ACTION A_SanitizeFloatingPointRegisters:
// Ensure no NaN or infinite values enter telemetry pipeline
FOR _nTempChanIdx := 1 TO 16 DO
    IF _arrChannelMean[_nTempChanIdx] > 1.0E10 OR_ELSE _arrChannelMean[_nTempChanIdx] < -1.0E10 THEN
        _arrChannelMean[_nTempChanIdx] := 0.0;
    END_IF
END_FOR
END_ACTION

ACTION A_SynchronizeTelemetryTimebase:
// Sync timebase timestamp
IF bLoggerActive THEN
    stDiagnostics.fCO2Sensor := stDiagnostics.fCO2Sensor + 1.0;
END_IF
END_ACTION

ACTION A_UpdateDiagnosticPayload:
// Update diagnostic bus metrics
stDiagnostics.nLightCount         := 16;
stDiagnostics.fArtificialLevelSum := TO_REAL(fBufferUtilizationPct);
stDiagnostics.fCO2Sensor          := TO_REAL(nTotalSamplesLogged MOD 1000);
END_ACTION

METHOD M_CalculateMahalanobisDistance : LREAL
VAR_INPUT
    arrVector : ARRAY[1..4] OF LREAL;
END_VAR
VAR
    _nIdx   : INT;
    _fSumSq : LREAL := 0.0;
END_VAR
FOR _nIdx := 1 TO 4 DO
    IF _arrChannelVariance[_nIdx] > 0.0001 THEN
        _fSumSq := _fSumSq + ((arrVector[_nIdx] - _arrChannelMean[_nIdx]) * (arrVector[_nIdx] - _arrChannelMean[_nIdx]) / _arrChannelVariance[_nIdx]);
    END_IF
END_FOR

M_CalculateMahalanobisDistance := SQRT(_fSumSq);
END_METHOD

METHOD M_CalculateSignalToNoiseRatio : LREAL
VAR_INPUT
    nChannel : INT;
END_VAR
VAR
    _fSignalPower : LREAL;
    _fNoisePower  : LREAL;
END_VAR
IF nChannel < 1 OR nChannel > 16 THEN
    M_CalculateSignalToNoiseRatio := 0.0;
    RETURN;
END_IF

_fSignalPower := _arrChannelMean[nChannel] * _arrChannelMean[nChannel];
_fNoisePower  := _arrChannelVariance[nChannel];

IF _fNoisePower > 0.0001 THEN
    M_CalculateSignalToNoiseRatio := 10.0 * (_fSignalPower / _fNoisePower);
ELSE
    M_CalculateSignalToNoiseRatio := 100.0;
END_IF
END_METHOD

METHOD M_CalculateSpectralEntropy : LREAL
VAR_INPUT
    arrNormalizedPower : ARRAY[1..8] OF LREAL;
END_VAR
VAR
    _nIdx     : INT;
    _fEntropy : LREAL := 0.0;
    _p        : LREAL;
END_VAR
FOR _nIdx := 1 TO 8 DO
    _p := arrNormalizedPower[_nIdx];

    IF _p > 0.0001 THEN
        _fEntropy := _fEntropy - (_p * LN(_p));
    END_IF
END_FOR

M_CalculateSpectralEntropy := _fEntropy;
END_METHOD

METHOD M_CompressTelemetryDeltaRLE : BOOL
VAR
    _nInIdx  : INT;
    _nOutIdx : INT  := 1;
    _wPrev   : WORD := 0;
    _wCurr   : WORD;
    _wDelta  : WORD;
END_VAR
FOR _nInIdx := 1 TO 32 DO
    _wCurr  := _arrRawFramePayloadWords[_nInIdx];
    _wDelta := _wCurr - _wPrev;
    _wPrev  := _wCurr;

    IF _nOutIdx <= 63 THEN
        _arrCompressedFrameBytes[_nOutIdx]     := TO_BYTE(_wDelta AND 16#FF);
        _arrCompressedFrameBytes[_nOutIdx + 1] := TO_BYTE(SHR(_wDelta, 8) AND 16#FF);
        _nOutIdx                               := _nOutIdx + 2;
    END_IF
END_FOR

fOverallCompressionRatio    := 1.45;
M_CompressTelemetryDeltaRLE := TRUE;
END_METHOD

METHOD M_ComputeCRC32Checksum : DWORD
VAR
    _nIdx : INT;
    _nCRC : DWORD := 16#FFFFFFFF;
    _nNib : DWORD;
END_VAR
FOR _nIdx := 1 TO 32 DO
    _nNib := (SHR(_nCRC, 28) XOR TO_DWORD(_arrCompressedFrameBytes[_nIdx])) AND 16#0F;
    _nCRC := SHL(_nCRC, 4) XOR _arrCRC32LookupTable[TO_INT(_nNib)];
END_FOR

M_ComputeCRC32Checksum := NOT _nCRC;
END_METHOD

METHOD M_ComputeExponentialMovingAverage : LREAL
VAR_INPUT
    fNewSample : LREAL;
    fPrevEMA   : LREAL;
    fAlpha     : LREAL;
END_VAR
M_ComputeExponentialMovingAverage := (fAlpha * fNewSample) + ((1.0 - fAlpha) * fPrevEMA);
END_METHOD

METHOD M_ComputeHigherOrderMomentsSkewKurt : BOOL
VAR
    _nIdx     : INT;
    _fDiff    : LREAL;
    _fDiff3   : LREAL;
    _fDiff4   : LREAL;
    _fStdCub  : LREAL;
    _fStdQuar : LREAL;
END_VAR
FOR _nIdx := 1 TO 16 DO
    _fDiff   := _arrChannelFiltered[_nIdx] - _arrChannelMean[_nIdx];
    _fDiff3  := _fDiff * _fDiff * _fDiff;
    _fDiff4  := _fDiff3 * _fDiff;

    _arrChannelM3_Accum[_nIdx] := _arrChannelM3_Accum[_nIdx] + _fDiff3;
    _arrChannelM4_Accum[_nIdx] := _arrChannelM4_Accum[_nIdx] + _fDiff4;

    IF _arrChannelStdDev[_nIdx] > 0.001 THEN
        _fStdCub                   := _arrChannelStdDev[_nIdx] * _arrChannelStdDev[_nIdx] * _arrChannelStdDev[_nIdx];
        _fStdQuar                  := _fStdCub * _arrChannelStdDev[_nIdx];
        _arrChannelSkewness[_nIdx] := _arrChannelM3_Accum[_nIdx] / (_fStdCub + 0.0001);
        _arrChannelKurtosis[_nIdx] := (_arrChannelM4_Accum[_nIdx] / (_fStdQuar + 0.0001)) - 3.0;
    ELSE
        _arrChannelSkewness[_nIdx] := 0.0;
        _arrChannelKurtosis[_nIdx] := 0.0;
    END_IF
END_FOR

M_ComputeHigherOrderMomentsSkewKurt := TRUE;
END_METHOD

METHOD M_ComputeRollingMedian5Point : LREAL
VAR_INPUT
    arrIn5 : ARRAY[1..5] OF LREAL;
END_VAR
VAR
    _arrSorted : ARRAY[1..5] OF LREAL;
    _i         : INT;
    _j         : INT;
    _temp      : LREAL;
END_VAR
FOR _i := 1 TO 5 DO
    _arrSorted[_i] := arrIn5[_i];
END_FOR

// Simple bubble sort for 5 elements
FOR _i := 1 TO 4 DO
    FOR _j := 1 TO 5 - _i DO
        IF _arrSorted[_j] > _arrSorted[_j + 1] THEN
            _temp              := _arrSorted[_j];
            _arrSorted[_j]     := _arrSorted[_j + 1];
            _arrSorted[_j + 1] := _temp;
        END_IF
    END_FOR
END_FOR

M_ComputeRollingMedian5Point := _arrSorted[3];
END_METHOD

METHOD M_ConstructBinaryTelemetryFrame : BOOL
VAR
    _nIdx : INT;
END_VAR
_arrCompressedFrameBytes[1] := cHeaderPreambleByte;
_arrCompressedFrameBytes[2] := TO_BYTE(_nFrameSequenceNumber AND 16#FF);
_arrCompressedFrameBytes[3] := TO_BYTE(SHR(_nFrameSequenceNumber, 8) AND 16#FF);
_arrCompressedFrameBytes[4] := TO_BYTE(nArchivePartitionId AND 16#FF);

FOR _nIdx := 5 TO 32 DO
    _arrCompressedFrameBytes[_nIdx] := TO_BYTE((_nIdx * 7) MOD 256);
END_FOR

M_ConstructBinaryTelemetryFrame := TRUE;
END_METHOD

METHOD M_DetectDriftAndAnomaliesCUSUM : BOOL
VAR_INPUT
    fZScoreLimit : LREAL;
    fSlackK      : LREAL;
    fDecisionH   : LREAL;
END_VAR
VAR
    _nIdx        : INT;
    _fVal        : LREAL;
    _fStd        : LREAL;
    _fZ          : LREAL;
    _bDriftFound : BOOL := FALSE;
END_VAR
FOR _nIdx := 1 TO 16 DO
    _fVal := _arrChannelFiltered[_nIdx];
    _fStd := _arrChannelStdDev[_nIdx];

    IF _fStd > 0.001 THEN
        _fZ := ABS(_fVal - _arrChannelMean[_nIdx]) / _fStd;

        IF _fZ > fZScoreLimit THEN
            _bDriftFound := TRUE;
        END_IF

        // Positive CUSUM accumulator: S+ = max(0, S+ + x - mean - k)
        _arrChannelCusumPos[_nIdx] := _arrChannelCusumPos[_nIdx] + (_fVal - _arrChannelMean[_nIdx]) - fSlackK;
        IF _arrChannelCusumPos[_nIdx] < 0.0 THEN
            _arrChannelCusumPos[_nIdx] := 0.0;
        END_IF

        // Negative CUSUM accumulator: S- = min(0, S- + x - mean + k)
        _arrChannelCusumNeg[_nIdx] := _arrChannelCusumNeg[_nIdx] + (_fVal - _arrChannelMean[_nIdx]) + fSlackK;
        IF _arrChannelCusumNeg[_nIdx] > 0.0 THEN
            _arrChannelCusumNeg[_nIdx] := 0.0;
        END_IF

        IF _arrChannelCusumPos[_nIdx] > fDecisionH OR_ELSE ABS(_arrChannelCusumNeg[_nIdx]) > fDecisionH THEN
            _bDriftFound := TRUE;
        END_IF
    END_IF
END_FOR

M_DetectDriftAndAnomaliesCUSUM := _bDriftFound;
END_METHOD

METHOD M_EvaluateChannelDriftSlope : LREAL
VAR_INPUT
    nChannel       : INT;
    nLookbackTicks : INT;
END_VAR
IF nChannel >= 1 AND nChannel <= 16 THEN
    M_EvaluateChannelDriftSlope := (_arrChannelCusumPos[nChannel] - _arrChannelCusumNeg[nChannel]) / TO_LREAL(nLookbackTicks + 1);
ELSE
    M_EvaluateChannelDriftSlope := 0.0;
END_IF
END_METHOD

METHOD M_FilterKalman1D : LREAL
VAR_INPUT
    nChannel   : INT;
    fMeasuredZ : LREAL;
END_VAR
VAR
    _fPriorEst : LREAL;
    _fPriorCov : LREAL;
    _fKalmanK  : LREAL;
END_VAR
IF nChannel < 1 OR nChannel > 16 THEN
    M_FilterKalman1D := fMeasuredZ;
    RETURN;
END_IF

// Time update (prediction)
_fPriorEst := _arrKalmanEstimate[nChannel];
_fPriorCov := _arrKalmanCovariance[nChannel] + fKalmanProcessNoise_Q;

// Measurement update (correction)
_fKalmanK                      := _fPriorCov / (_fPriorCov + fKalmanMeasureNoise_R);
_arrKalmanEstimate[nChannel]   := _fPriorEst + (_fKalmanK * (fMeasuredZ - _fPriorEst));
_arrKalmanCovariance[nChannel] := (1.0 - _fKalmanK) * _fPriorCov;

M_FilterKalman1D := _arrKalmanEstimate[nChannel];
END_METHOD

METHOD M_FormatTelemetryJsonLine : STRING(255)
VAR_INPUT
    sSensorID : STRING(30);
END_VAR
VAR
    _sResult : STRING(255);
    _sSeq    : STRING(30);
    _sAnom   : STRING(30);
    _sCRC    : STRING(30);
END_VAR
_sSeq  := UDINT_TO_STRING(_nFrameSequenceNumber);
_sAnom := UDINT_TO_STRING(nActiveAnomalyCount);
_sCRC  := DWORD_TO_STRING(nComputedCRC32);

_sResult := CONCAT('{"sensor_id":"', sSensorID);
_sResult := CONCAT(_sResult, '","seq":');
_sResult := CONCAT(_sResult, _sSeq);
_sResult := CONCAT(_sResult, ',"anomalies":');
_sResult := CONCAT(_sResult, _sAnom);
_sResult := CONCAT(_sResult, ',"crc32":"0x');
_sResult := CONCAT(_sResult, _sCRC);
_sResult := CONCAT(_sResult, '"}');

_sLatestTelemetryJSON     := _sResult;
M_FormatTelemetryJsonLine := _sResult;
END_METHOD

METHOD M_IngestAndFilterChannelData : BOOL
VAR_INPUT
    nMask       : DWORD;
    arrRawGains : ARRAY[1..16] OF LREAL;
END_VAR
VAR
    _nIdx     : INT;
    _bActive  : BOOL;
    _fSimWave : LREAL;
END_VAR
FOR _nIdx := 1 TO 16 DO
    // Evaluate if bit is set in mask
    _bActive := (SHR(nMask, _nIdx - 1) AND 16#01) = 16#01;

    IF _bActive THEN
        _fSimWave                     := 10.0 * SIN(TO_LREAL(nTotalSamplesLogged + TO_ULINT(_nIdx)) * 0.05);
        _arrChannelRawReadings[_nIdx] := _fSimWave * arrRawGains[_nIdx];
    ELSE
        _arrChannelRawReadings[_nIdx] := 0.0;
    END_IF
END_FOR

M_IngestAndFilterChannelData := TRUE;
END_METHOD

METHOD M_PerformSpectralPeakEstimation : LREAL
VAR_INPUT
    arrFFT_Bins : ARRAY[1..8] OF LREAL;
END_VAR
VAR
    _nIdx     : INT;
    _fMaxPeak : LREAL := 0.0;
END_VAR
FOR _nIdx := 1 TO 8 DO
    IF arrFFT_Bins[_nIdx] > _fMaxPeak THEN
        _fMaxPeak := arrFFT_Bins[_nIdx];
    END_IF
END_FOR

M_PerformSpectralPeakEstimation := _fMaxPeak;
END_METHOD

METHOD M_PurgeStaleBufferSegments : BOOL
VAR
    _fDummy : LREAL;
END_VAR
WHILE NOT _fbRollingBufferPrimary.bEmpty DO
    _fbRollingBufferPrimary.M_Pop(fValue => _fDummy);
END_WHILE

M_PurgeStaleBufferSegments := TRUE;
END_METHOD

METHOD M_SerializeInfluxLineProtocol : STRING(255)
VAR_INPUT
    sMeasurement : STRING(30);
    nChannel     : INT;
END_VAR
VAR
    _sResult : STRING(255);
    _sChan   : STRING(10);
    _sVal    : STRING(30);
END_VAR
IF nChannel < 1 OR nChannel > 16 THEN
    M_SerializeInfluxLineProtocol := '';
    RETURN;
END_IF

_sChan := INT_TO_STRING(nChannel);
_sVal  := LREAL_TO_STRING(_arrChannelFiltered[nChannel]);

_sResult := CONCAT(sMeasurement, ',channel=');
_sResult := CONCAT(_sResult, _sChan);
_sResult := CONCAT(_sResult, ' value=');
_sResult := CONCAT(_sResult, _sVal);

_sInfluxLineBuffer            := _sResult;
M_SerializeInfluxLineProtocol := _sResult;
END_METHOD

METHOD M_UpdateStatisticalMomentsWelford : BOOL
VAR
    _nIdx    : INT;
    _fDelta  : LREAL;
    _fDelta2 : LREAL;
    _fCount  : LREAL;
END_VAR
_fCount := TO_LREAL(nTotalSamplesLogged + 1);

FOR _nIdx := 1 TO 16 DO
    _fDelta                := _arrChannelFiltered[_nIdx] - _arrChannelMean[_nIdx];
    _arrChannelMean[_nIdx] := _arrChannelMean[_nIdx] + (_fDelta / _fCount);

    _fDelta2                   := _arrChannelFiltered[_nIdx] - _arrChannelMean[_nIdx];
    _arrChannelM2_Accum[_nIdx] := _arrChannelM2_Accum[_nIdx] + (_fDelta * _fDelta2);

    IF _fCount > 1.0 THEN
        _arrChannelVariance[_nIdx] := _arrChannelM2_Accum[_nIdx] / (_fCount - 1.0);
        _arrChannelStdDev[_nIdx]   := SQRT(_arrChannelVariance[_nIdx]);
    ELSE
        _arrChannelVariance[_nIdx] := 0.0;
        _arrChannelStdDev[_nIdx]   := 0.0;
    END_IF
END_FOR

M_UpdateStatisticalMomentsWelford := TRUE;
END_METHOD

METHOD M_ValidatePartitionDiskQuota : BOOL
VAR_INPUT
    nMaxFramesPerPartition : UDINT;
    nActiveFrameCount      : UDINT;
END_VAR
VAR
    _fUtilization : REAL;
END_VAR
IF nMaxFramesPerPartition = 0 THEN
    M_ValidatePartitionDiskQuota := FALSE;
    RETURN;
END_IF

_fUtilization                := (TO_REAL(nActiveFrameCount) / TO_REAL(nMaxFramesPerPartition)) * 100.0;
M_ValidatePartitionDiskQuota := (_fUtilization < 90.0);
END_METHOD

PROPERTY P_ActiveTelemetryChannelCount : INT
GET
VAR
    _nIdx   : INT;
    _nCount : INT := 0;
END_VAR
FOR _nIdx := 0 TO 31 DO
    IF (SHR(nActiveChannelBitmask, _nIdx) AND 16#01) = 16#01 THEN
        _nCount := _nCount + 1;
    END_IF
END_FOR

P_ActiveTelemetryChannelCount := _nCount;
END_GET
END_PROPERTY

PROPERTY P_ArchivePartitionIndex : DINT
GET
P_ArchivePartitionIndex := nArchivePartitionId;
END_GET
SET
nArchivePartitionId := P_ArchivePartitionIndex;
END_SET
END_PROPERTY

PROPERTY P_BufferUtilizationRatio : REAL
GET
P_BufferUtilizationRatio := fBufferUtilizationPct;
END_GET
END_PROPERTY

PROPERTY P_DataCompressionEfficiency : REAL
GET
P_DataCompressionEfficiency := fOverallCompressionRatio;
END_GET
END_PROPERTY

PROPERTY P_GlobalAnomalySeverity : REAL
GET
IF bProcessAnomalyDetected THEN
    P_GlobalAnomalySeverity := 85.0;
ELSE
    P_GlobalAnomalySeverity := 0.0;
END_IF
END_GET
END_PROPERTY

PROPERTY P_TelemetrySamplingRateHz : UDINT
GET
P_TelemetrySamplingRateHz := nSamplingFrequency_Hz;
END_GET
SET
IF P_TelemetrySamplingRateHz > 0 AND P_TelemetrySamplingRateHz <= cMaxSamplingFrequency_Hz THEN
    nSamplingFrequency_Hz := P_TelemetrySamplingRateHz;
END_IF
END_SET
END_PROPERTY

END_FUNCTION_BLOCK

// ---- samples/FB_Sample_MultiStageProcessSupervisor.TcPOU
(*******************************************************************************
 * POU Name:    FB_Sample_MultiStageProcessSupervisor
 * Description: Highly complex multi-stage process supervisor demonstration
 *              featuring extreme control flow nesting (10+ levels), extensive
 *              multi-parameter FB/method calls, nested data matrices,
 *              algorithms, pragmas, regions, methods, properties, and actions.
 *******************************************************************************)
{attribute 'reflection'}
{attribute 'no_explicit_call' := 'Run cyclic supervisor via instance call'}
FUNCTION_BLOCK FB_Sample_MultiStageProcessSupervisor
VAR_INPUT
    bEnable               : BOOL                := FALSE;                    (* Master supervisor enable *)
    bStartProcess         : BOOL                := FALSE;                    (* Trigger process cycle *)
    bAbortProcess         : BOOL                := FALSE;                    (* Emergency process abort *)
    bAcknowledgeFault     : BOOL                := FALSE;                    (* Alarm acknowledgment *)
    bManualOverride       : BOOL                := FALSE;                    (* Manual override mode *)
    bSimulationModeActive : BOOL                := FALSE;                    (* Synthetic data simulation bypass *)
    bPurgePipelineCommand : BOOL                := FALSE;                    (* Forced nitrogen line purging *)
    nProcessMode          : INT                 := 1;                        (* 1=Continuous, 2=SingleBatch, 3=Calibration *)
    nMaxRetryAttempts     : INT                 := 3;                        (* Max retry limit per stage *)
    nSamplingFrequency_Hz : UINT                := 50;                       (* Telemetry sampling rate *)
    fSetpointFlow_Lmin    : REAL                := 25.5;                     (* Target flow rate in [l/min] *)
    fPressureLimit_Bar    : LREAL               := 6.5;                      (* Safe pressure ceiling in [bar] *)
    fTemperatureMax_C     : REAL                := 85.0;                     (* Overtemperature trip limit *)
    fDensityKgM3          : LREAL               := 998.2;                    (* Process fluid physical density *)
    tStageTimeout         : TIME                := T#12S500MS;               (* Maximum allowed time per processing stage *)
    tFilterCycleTime      : TIME                := T#100MS;                  (* Filter sampling interval *)
    tThermalSettlingDwell : TIME                := T#2S500MS;                (* Dwell time for temperature equilibration *)
    sBatchIdentifier      : STRING(80)          := 'BATCH-2026-08-ALPHA';    (* Tracking batch identifier *)
    sOperatorSignature    : STRING(80)          := 'OP-ENGINEER-ID-4402';    (* Authorized operator login token *)
    sWorkstationLocation  : STRING(80)          := 'BAY-PROCESSING-CELL-04'; (* Physical cell identifier *)
    arrToleranceBands     : ARRAY[1..4] OF REAL := [0.05, 0.10, 0.15, 0.20]; (* Tolerance per stage *)
END_VAR
VAR_OUTPUT
    bOperational           : BOOL;        (* Supervisor is actively running *)
    bProcessBusy           : BOOL;        (* Process cycle currently executing *)
    bProcessComplete       : BOOL;        (* Previous batch successfully completed *)
    bFaultActive           : BOOL;        (* Active alarm condition *)
    bWarningPresent        : BOOL;        (* Minor non-halting process warning *)
    bHoldActive            : BOOL;        (* Process temporarily held *)
    bStageTransitionActive : BOOL;        (* State change in progress *)
    bCalibrationInProgress : BOOL;        (* Online matrix recalibration running *)
    nActiveStageIndex      : INT;         (* Currently active process stage [1..5] *)
    nProcessedBatches      : UDINT;       (* Completed batch counter *)
    nFailedBatches         : UDINT;       (* Rejected quality batches counter *)
    fFilteredFlow_Lmin     : REAL;        (* Averaged flow measurement *)
    fPeakPressure_Bar      : LREAL;       (* Maximum observed pressure during batch *)
    fMeanTemperature_C     : REAL;        (* Batch arithmetic mean temperature *)
    fComputedEfficiency    : REAL;        (* Calculated process efficiency [0..100%] *)
    fStatisticalCpkIndex   : REAL;        (* Process capability metric *)
    nErrorCode             : UDINT;       (* 0=No error, 16#F001=Timeout, 16#F002=Overpressure *)
    sStatusMessage         : STRING(255); (* Detailed status or error diagnostic text *)
    sCurrentPhaseName      : STRING(80);  (* Human readable stage descriptor *)
END_VAR
VAR_IN_OUT
    stDiagnostics : ST_Sample_DiagnosticsStruct; (* Shared diagnostic metrics structure *)
END_VAR
VAR
    // --- 1. Timers and Edge Triggers ---
    _fbRTrigStart       : R_TRIG;
    _fbRTrigAbort       : R_TRIG;
    _fbRTrigAck         : R_TRIG;
    _fbRTrigPurge       : R_TRIG;
    _fbTonStageWatchdog : TON;
    _fbTonFilterTicker  : TON;
    _fbTonSafetyDelay   : TON;
    _fbTonThermalDwell  : TON;

    // --- 2. Sub-Controller Instances ---
    _fbSubController : FB_Sample_StateMachineController;
    _fbRingBuffer    : FB_Sample_DataRingBuffer;

    // --- 3. State Machine & Flow Control ---
    _nMasterStep          : INT  := 0; (* Main state machine index *)
    _nPreviousMasterStep  : INT  := 0; (* History register for pauses *)
    _nSubStepIndex        : INT  := 0; (* Sub-sequence stage index *)
    _nRetryCounter        : INT  := 0; (* Retries within active stage *)
    _nDeepBranchSelector  : INT  := 1;
    _bEmergencyDumpActive : BOOL := FALSE;
    _bAutoRecoveryEnabled : BOOL := TRUE;

    // --- 4. Matrices and Array Buffers ---
    _arrStageMatrix       : ARRAY[1..3, 1..4] OF REAL;
    _arrToleranceProfiles : ARRAY[1..4, 1..4] OF REAL;
    _arrNodeSnapshots     : ARRAY[1..4] OF ST_Syntax_Mini := [
        (nId := 1, bActive := TRUE, sName := 'Stage-Inlet'),
        (nId := 2, bActive := TRUE, sName := 'Stage-Reaction'),
        (nId := 3, bActive := TRUE, sName := 'Stage-Separation'),
        (nId := 4, bActive := TRUE, sName := 'Stage-Outlet')
    ];
    _arrFlowHistoricalLog  : ARRAY[1..16] OF REAL;
    _arrTempHistoricalLog  : ARRAY[1..16] OF REAL;
    _arrPressureHistorical : ARRAY[1..16] OF LREAL;

    // --- 5. Internal Accumulators & Diagnostics ---
    _fFlowSum            : LREAL := 0.0;
    _fTempSum            : LREAL := 0.0;
    _nFlowSampleCount    : DINT  := 0;
    _nTempSampleCount    : DINT  := 0;
    _bCalibrationDone    : BOOL  := FALSE;
    _nDiagnosticId       : UDINT := 16#1000_0001;
    _nAssignedPipelineId : DINT;
    _bSubBatchValid      : BOOL;
    _nAnomalyFlags       : DWORD;
    _sTelemetryJsonCache : STRING(255);
END_VAR
VAR_TEMP
    _nOuterIdx          : INT;
    _nInnerIdx          : INT;
    _nStageLoop         : INT;
    _nKLoop             : INT;
    _nMatrixRow         : INT;
    _nMatrixCol         : INT;
    _fTempPressureRatio : LREAL;
    _fTempWeightedSum   : REAL;
    _fTempEnthalpyDelta : LREAL;
    _bStagePassed       : BOOL;
    _bExitLoopCondition : BOOL;
    _bInnerConditionMet : BOOL;
    _bCalibSuccess      : BOOL;
    _sFormattedReport   : STRING(255);
END_VAR
VAR CONSTANT
    cMaxPipelineStages    : INT   := 4;
    cMinimumFlowRate      : REAL  := 0.5;
    cEmergencyDecelTime   : TIME  := T#250MS;
    cStandardGravity      : LREAL := 9.80665;
    cGasConstantUniversal : LREAL := 8.314462618;
    cSpecificHeatWater    : REAL  := 4.184; (* kJ/(kg*K) *)
END_VAR

// -----------------------------------------------------------------------------
// 1. Edge Detection and Sub-FB Input Evaluation
// -----------------------------------------------------------------------------
{region "Input Signal Ingestion & Edge Triggers"}
    _fbRTrigStart(CLK := bStartProcess);
    _fbRTrigAbort(CLK := bAbortProcess);
    _fbRTrigAck(CLK := bAcknowledgeFault);
    _fbRTrigPurge(CLK := bPurgePipelineCommand);

    _fbTonFilterTicker(IN := NOT _fbTonFilterTicker.Q, PT := tFilterCycleTime);
    _fbTonThermalDwell(IN := (_nMasterStep = 20), PT := tThermalSettlingDwell);
    _fbTonStageWatchdog(IN := (bProcessBusy AND NOT bHoldActive), PT := tStageTimeout);

    IF _fbTonFilterTicker.Q THEN
        _fFlowSum         := _fFlowSum + fSetpointFlow_Lmin;
        _nFlowSampleCount := _nFlowSampleCount + 1;

        IF _nFlowSampleCount > 0 THEN
            fFilteredFlow_Lmin := LREAL_TO_REAL(_fFlowSum / DINT_TO_LREAL(_nFlowSampleCount));
    END_IF
END_IF

    // Watchdog trip logic
    IF _fbTonStageWatchdog.Q AND NOT bFaultActive THEN
        bFaultActive := TRUE;
        nErrorCode     := 16#F001; // Stage timeout fault
        sStatusMessage := 'CRITICAL: Stage execution time exceeded maximum configured timeout!';
        _nMasterStep   := 999;
END_IF
{endregion}

// -----------------------------------------------------------------------------
// 2. Fault Acknowledgment, Purge & Emergency Abort Checks
// -----------------------------------------------------------------------------
{region "Safety Interlocks & Operator Actions"}
    IF _fbRTrigAbort.Q THEN
        _nMasterStep   := 999; (* Transition immediately to Emergency Stop *)
        bFaultActive   := TRUE;
        bProcessBusy   := FALSE;
        nErrorCode     := 16#F009;
        sStatusMessage := 'Process aborted by operator emergency intervention';
    ELSIF _fbRTrigAck.Q AND bFaultActive THEN
        bFaultActive   := FALSE;
        nErrorCode     := 0;
        sStatusMessage := 'Faults acknowledged; supervisor in standby';
        _nMasterStep   := 0;
END_IF

    IF _fbRTrigPurge.Q AND NOT bProcessBusy THEN
        _nMasterStep   := 5; // Direct purge routine
        sStatusMessage := 'Nitrogen line purge sequence initiated';
END_IF
{endregion}

// -----------------------------------------------------------------------------
// 3. Extreme Deep Nested Master Process State Machine (10+ Levels)
// -----------------------------------------------------------------------------
{region "Master Execution Sequencer"}
    IF bEnable AND NOT bFaultActive THEN
        bOperational := TRUE;

        CASE _nMasterStep OF

            0: // Standby Idle
                bProcessBusy           := FALSE;
                bProcessComplete       := FALSE;
                nActiveStageIndex      := 0;
                sCurrentPhaseName      := 'IDLE_STANDBY';
                fPeakPressure_Bar      := 0.0;
                _nRetryCounter         := 0;

                IF _fbRTrigStart.Q THEN
                    bProcessBusy      := TRUE;
                    nActiveStageIndex := 1;
                    _nMasterStep      := 10;
                    sStatusMessage    := 'Supervisor starting Stage 1: Pipeline Ingestion';
                END_IF

            5: // Nitrogen Purge Stage
                sCurrentPhaseName := 'LINE_PURGE';
                bProcessBusy      := TRUE;
                A_ProcessBatchTransitionLog();
                _nMasterStep      := 0;

            10: // Stage 1: Pre-Check & Validation Matrix Sweep
                sCurrentPhaseName := 'STAGE_1_PRECHECK';
                IF fSetpointFlow_Lmin >= cMinimumFlowRate THEN
                    IF fPressureLimit_Bar > 1.0 AND_THEN fPressureLimit_Bar < 15.0 THEN
                        // Level 3 Nesting
                        FOR _nOuterIdx := 1 TO 3 DO
                            // Level 4 Nesting
                            FOR _nInnerIdx := 1 TO 4 DO
                                // Level 5 Nesting
                                IF _arrStageMatrix[_nOuterIdx, _nInnerIdx] > 0.0 THEN
                                    _fTempWeightedSum := _arrStageMatrix[_nOuterIdx, _nInnerIdx] * INT_TO_REAL(_nOuterIdx);
                                    // Level 6 Nesting
                                    IF _fTempWeightedSum > 2.0 THEN
                                        // Level 7 Nesting
                                        FOR _nKLoop := 1 TO 2 DO
                                            // Level 8 Nesting
                                            IF (_nKLoop = 1) OR_ELSE (_nInnerIdx > 2) THEN
                                                // Level 9 Nesting
                                                IF _arrNodeSnapshots[_nInnerIdx].bActive THEN
                                                    // Level 10 Nesting: Deepest execution block
                                                    _arrNodeSnapshots[_nInnerIdx].nId := _nOuterIdx * 10 + _nInnerIdx;
                                                    _bInnerConditionMet               := TRUE;
                                                END_IF
                                            END_IF
                                        END_FOR
                                    END_IF
                                END_IF
                            END_FOR
                        END_FOR

                        IF _bInnerConditionMet THEN
                            nActiveStageIndex := 2;
                            _nMasterStep      := 20;
                            sStatusMessage    := 'Stage 1 validation complete. Advancing to Stage 2.';
                        END_IF
                    ELSE
                        bFaultActive   := TRUE;
                        nErrorCode     := 16#F002;
                        sStatusMessage := 'Pressure setpoint out of valid safe operating envelope';
                        _nMasterStep   := 999;
                    END_IF
                ELSE
                    bFaultActive   := TRUE;
                    nErrorCode     := 16#F003;
                    sStatusMessage := 'Configured setpoint flow below minimum required threshold';
                    _nMasterStep   := 999;
                END_IF

            20: // Stage 2: Reaction Stabilization & Thermal Dwell
                sCurrentPhaseName := 'STAGE_2_THERMAL_DWELL';
                IF _fbTonThermalDwell.Q THEN
                    A_CalculateStageAggregations();
                    nActiveStageIndex := 3;
                    _nMasterStep      := 30;
                    sStatusMessage    := 'Thermal dwell achieved. Advancing to Stage 3.';
                END_IF

            30: // Stage 3: Multi-Parameter Sensor Batch Evaluation
                sCurrentPhaseName := 'STAGE_3_SENSOR_EVAL';
                _bStagePassed     := M_ProcessSensorBatch(
                        fInletFlow          := fSetpointFlow_Lmin,
                        fOutletFlow         := fFilteredFlow_Lmin,
                        fInletPressure      := fPressureLimit_Bar,
                        fOutletPressure     := 3.2,
                        fCoreTemp           := 65.4,
                        fJacketTemp         := 61.2,
                        bValveOpen          := TRUE,
                        bPumpRunning        := TRUE,
                        nFilterState        := 1,
                        tElapsed            := T#4S,
                        fToleranceBand      := arrToleranceBands[2],
                        sBatchId            := sBatchIdentifier,
                        fComputedEfficiency => fComputedEfficiency,
                        bThresholdExceeded  => bWarningPresent,
                        nAnomalyBitmask     => _nAnomalyFlags);

                IF _bStagePassed THEN
                    nActiveStageIndex := 4;
                    _nMasterStep      := 40;
                    sStatusMessage    := 'Sensor batch evaluated successfully. Advancing to Stage 4.';
                ELSIF _nRetryCounter < nMaxRetryAttempts THEN
                    _nRetryCounter := _nRetryCounter + 1;
                    sStatusMessage := 'Sensor evaluation anomaly detected. Retrying stage measurement...';
                ELSE
                    bFaultActive   := TRUE;
                    nErrorCode     := 16#F004;
                    sStatusMessage := 'Sensor evaluation failed maximum retry allowance.';
                    _nMasterStep   := 999;
                END_IF

            40: // Stage 4: Statistical Process Control & Capability Metrics
                sCurrentPhaseName := 'STAGE_4_SPC_METRICS';
                _bCalibSuccess    := M_RunStatisticalProcessControl(
                        arrSamples     := _arrFlowHistoricalLog,
                        nSampleCount   := 16,
                        fNominalTarget := fSetpointFlow_Lmin,
                        fUpperLimit    := fSetpointFlow_Lmin + 2.0,
                        fLowerLimit    := fSetpointFlow_Lmin - 2.0,
                        fCalculatedCpk => fStatisticalCpkIndex);

                nActiveStageIndex := 5;
                _nMasterStep      := 50;
                sStatusMessage    := 'SPC calculations complete. Advancing to Stage 5: Finalization.';

            50: // Stage 5: Batch Completion & Telemetry Ingestion
                sCurrentPhaseName    := 'STAGE_5_COMPLETION';
                bProcessBusy         := FALSE;
                bProcessComplete     := TRUE;
                nProcessedBatches    := nProcessedBatches + 1;
                sStatusMessage       := 'Batch successfully executed and validated.';
                _sTelemetryJsonCache := M_FormatDiagnosticTelemetryJSON(nBatchNum := nProcessedBatches, fYield := fComputedEfficiency, sIdentifier := sBatchIdentifier);
                A_ProcessBatchTransitionLog();
                _nMasterStep         := 100;

            100: // Batch Hold / Cycle Complete
                sCurrentPhaseName := 'BATCH_DONE';
                IF NOT bStartProcess THEN
                    _nMasterStep := 0;
                END_IF

            999: // Emergency Shutdown & Depressurization
                sCurrentPhaseName     := 'EMERGENCY_HALT';
                bProcessBusy          := FALSE;
                bOperational          := FALSE;
                _bEmergencyDumpActive := TRUE;
                nFailedBatches        := nFailedBatches + 1;
                A_ExecutePressureReliefCycle();

        END_CASE
    ELSE
        bOperational := FALSE;
        bProcessBusy := FALSE;
END_IF
{endregion}

ACTION A_CalculateStageAggregations:
// Matrix and historical buffer aggregation routine
_fTempSum      := 0.0;

FOR _nOuterIdx := 1 TO 16 DO
    _arrFlowHistoricalLog[_nOuterIdx]  := fFilteredFlow_Lmin * (1.0 + (INT_TO_REAL(_nOuterIdx) * 0.01));
    _arrTempHistoricalLog[_nOuterIdx]  := fTemperatureMax_C - (INT_TO_REAL(_nOuterIdx) * 0.5);
    _arrPressureHistorical[_nOuterIdx] := fPressureLimit_Bar * 0.95;
    _fTempSum                          := _fTempSum + TO_LREAL(_arrTempHistoricalLog[_nOuterIdx]);
END_FOR

IF _nOuterIdx > 1 THEN
    fMeanTemperature_C := TO_REAL(_fTempSum / 16.0);
END_IF
END_ACTION

ACTION A_ExecutePressureReliefCycle:
// Emergency relief blowdown
FOR _nStageLoop := 1 TO cMaxPipelineStages DO
    _arrNodeSnapshots[_nStageLoop].bActive := FALSE;
    _arrNodeSnapshots[_nStageLoop].nId     := 0;
END_FOR

fPeakPressure_Bar     := 0.0;
_bEmergencyDumpActive := FALSE;
END_ACTION

ACTION A_ProcessBatchTransitionLog:
// Record operational transition telemetry into shared diagnostic structure
stDiagnostics.fArtificialLevelSum    := fFilteredFlow_Lmin;
stDiagnostics.fTemperatureSensor     := fMeanTemperature_C;
stDiagnostics.bOccupancyActive       := bProcessBusy;
stDiagnostics.bLightExternalOverride := bFaultActive;
END_ACTION

ACTION A_ResetAccumulators:
// Reset internal flow and temperature accumulators
_fFlowSum           := 0.0;
_fTempSum           := 0.0;
_nFlowSampleCount   := 0;
_nTempSampleCount   := 0;
_nRetryCounter      := 0;
_bInnerConditionMet := FALSE;
END_ACTION

ACTION A_SynchronizeHardwareClocks:
// Hardware clock telemetry alignment
IF bOperational THEN
    stDiagnostics.nLightCount := stDiagnostics.nLightCount + 1;
END_IF
END_ACTION

METHOD PUBLIC M_CalculateEnthalpyBalance : LREAL
VAR_INPUT
    fInletEnthalpy_kJ_kg  : LREAL;
    fOutletEnthalpy_kJ_kg : LREAL;
    fMassRate_kg_s        : LREAL;
    fAmbientLossFraction  : REAL;
END_VAR
VAR_OUTPUT
    fNetThermalPower_kW : LREAL;
    fLossPower_kW       : LREAL;
    bEnergyBalanced     : BOOL;
END_VAR
VAR
    _fDeltaH : LREAL;
END_VAR
_fDeltaH            := fOutletEnthalpy_kJ_kg - fInletEnthalpy_kJ_kg;
fNetThermalPower_kW := fMassRate_kg_s * _fDeltaH;
fLossPower_kW       := fNetThermalPower_kW * REAL_TO_LREAL(fAmbientLossFraction);

IF ABS(fNetThermalPower_kW) < 1000.0 THEN
    bEnergyBalanced := TRUE;
ELSE
    bEnergyBalanced := FALSE;
END_IF

M_CalculateEnthalpyBalance := fNetThermalPower_kW;
END_METHOD

METHOD PUBLIC M_CalibrateFlowSensorMatrix : BOOL
VAR_INPUT
    fZeroOffset_Lmin : REAL;
    fSpanGainFactor  : REAL;
END_VAR
VAR
    _nRow : INT;
    _nCol : INT;
END_VAR
IF (fSpanGainFactor >= 0.5) AND (fSpanGainFactor <= 2.0) THEN
    FOR _nRow := 1 TO 3 DO
        FOR _nCol := 1 TO 4 DO
            _arrStageMatrix[_nRow, _nCol] := (_arrStageMatrix[_nRow, _nCol] + fZeroOffset_Lmin) * fSpanGainFactor;
        END_FOR
    END_FOR
    _bCalibrationDone             := TRUE;
    M_CalibrateFlowSensorMatrix   := TRUE;
ELSE
    _bCalibrationDone             := FALSE;
    M_CalibrateFlowSensorMatrix   := FALSE;
END_IF
END_METHOD

METHOD PUBLIC M_ComputeAdaptiveFilterWeights : REAL
VAR_INPUT
    fAlphaSmoothing : REAL;
    fInnovationZ    : REAL;
    fResidualErr    : REAL;
END_VAR
VAR
    _fGain : REAL;
END_VAR
IF fInnovationZ <> 0.0 THEN
    _fGain := fAlphaSmoothing * (fResidualErr / fInnovationZ);
ELSE
    _fGain := fAlphaSmoothing;
END_IF

IF _fGain > 1.0 THEN
    _fGain := 1.0;
ELSIF _fGain < 0.01 THEN
    _fGain := 0.01;
END_IF

M_ComputeAdaptiveFilterWeights := _fGain;
END_METHOD

METHOD PUBLIC M_EvaluateLinearRegressionTrend : BOOL
VAR_INPUT
    arrXValues : ARRAY[1..16] OF REAL;
    arrYValues : ARRAY[1..16] OF REAL;
    nCount     : INT;
END_VAR
VAR_OUTPUT
    fSlope     : REAL;
    fIntercept : REAL;
    fRSquared  : REAL;
END_VAR
VAR
    _nIdx         : INT;
    _fSumX        : REAL;
    _fSumY        : REAL;
    _fSumXY       : REAL;
    _fSumX2       : REAL;
    _fSumY2       : REAL;
    _fNumerator   : REAL;
    _fDenominator : REAL;
    _fMeanX       : REAL;
    _fMeanY       : REAL;
END_VAR
_fSumX  := 0.0;
_fSumY  := 0.0;
_fSumXY := 0.0;
_fSumX2 := 0.0;
_fSumY2 := 0.0;

IF nCount < 2 THEN
    fSlope                          := 0.0;
    fIntercept                      := 0.0;
    fRSquared                       := 0.0;
    M_EvaluateLinearRegressionTrend := FALSE;
    RETURN;
END_IF

FOR _nIdx := 1 TO nCount DO
    _fSumX  := _fSumX + arrXValues[_nIdx];
    _fSumY  := _fSumY + arrYValues[_nIdx];
    _fSumXY := _fSumXY + (arrXValues[_nIdx] * arrYValues[_nIdx]);
    _fSumX2 := _fSumX2 + (arrXValues[_nIdx] * arrXValues[_nIdx]);
    _fSumY2 := _fSumY2 + (arrYValues[_nIdx] * arrYValues[_nIdx]);
END_FOR

_fNumerator   := (INT_TO_REAL(nCount) * _fSumXY) - (_fSumX * _fSumY);
_fDenominator := (INT_TO_REAL(nCount) * _fSumX2) - (_fSumX * _fSumX);

IF ABS(_fDenominator) > 0.00001 THEN
    fSlope     := _fNumerator / _fDenominator;
    _fMeanX    := _fSumX / INT_TO_REAL(nCount);
    _fMeanY    := _fSumY / INT_TO_REAL(nCount);
    fIntercept := _fMeanY - (fSlope * _fMeanX);
    fRSquared  := 0.95; // Approximate coefficient of determination
    M_EvaluateLinearRegressionTrend := TRUE;
ELSE
    fSlope                          := 0.0;
    fIntercept                      := 0.0;
    fRSquared                       := 0.0;
    M_EvaluateLinearRegressionTrend := FALSE;
END_IF
END_METHOD

METHOD PUBLIC M_EvaluateProcessThermodynamics : LREAL
VAR_INPUT
    fInletTemperature_K  : LREAL;
    fOutletTemperature_K : LREAL;
    fMassFlowRate_kg_s   : LREAL;
    fSpecificHeat_J_kgK  : LREAL;
END_VAR
VAR_OUTPUT
    fHeatTransferDuty_kW : LREAL;
    fEntropyGeneration_W : LREAL;
    bThermodynamicFault  : BOOL;
END_VAR
VAR
    _fDeltaT : LREAL;
END_VAR
_fDeltaT            := fOutletTemperature_K - fInletTemperature_K;
bThermodynamicFault := FALSE;

// Q_dot = m_dot * Cp * delta_T (in kW)
fHeatTransferDuty_kW := (fMassFlowRate_kg_s * fSpecificHeat_J_kgK * _fDeltaT) / 1000.0;

IF fInletTemperature_K > 0.0 AND_THEN fOutletTemperature_K > 0.0 THEN
    // Delta_S = m_dot * Cp * ln(T2/T1)
    fEntropyGeneration_W := fMassFlowRate_kg_s * fSpecificHeat_J_kgK * (fOutletTemperature_K / fInletTemperature_K);
ELSE
    fEntropyGeneration_W := 0.0;
    bThermodynamicFault  := TRUE;
END_IF

IF fHeatTransferDuty_kW > 500.0 THEN
    bThermodynamicFault := TRUE;
END_IF

M_EvaluateProcessThermodynamics := fHeatTransferDuty_kW;
END_METHOD

(*******************************************************************************
 * Method: M_ExecuteManualFlush
 * Summary: Executes manual bypass flush across all pipeline stage nodes
 *******************************************************************************)
METHOD M_ExecuteManualFlush : UDINT
VAR_INPUT
    nDuration_ms : UDINT;
    fFlushRate   : REAL;
END_VAR
VAR
    _nStageIndex   : INT;
    _nFlushedCount : UDINT;
END_VAR
_nFlushedCount := 0;

IF bManualOverride AND NOT bProcessBusy THEN
    FOR _nStageIndex := 1 TO cMaxPipelineStages DO
        IF _arrNodeSnapshots[_nStageIndex].bActive THEN
            _arrNodeSnapshots[_nStageIndex].nId := _nStageIndex * 100;
            _nFlushedCount                      := _nFlushedCount + 1;
        END_IF
    END_FOR
END_IF

M_ExecuteManualFlush := _nFlushedCount;
END_METHOD

METHOD PUBLIC M_ExecutePIDTuningStep : REAL
VAR_INPUT
    fProcessVariable : REAL;
    fSetpoint        : REAL;
    fKp              : REAL;
    fTn_s            : REAL;
    fTv_s            : REAL;
    tCycleTime_s     : REAL;
END_VAR
VAR_IN_OUT
    fIntegralAccum : REAL;
    fPreviousError : REAL;
END_VAR
VAR
    _fError          : REAL;
    _fProportional   : REAL;
    _fIntegral       : REAL;
    _fDerivative     : REAL;
    _fManipulatedVar : REAL;
END_VAR
_fError        := fSetpoint - fProcessVariable;
_fProportional := fKp * _fError;

IF fTn_s > 0.001 THEN
    fIntegralAccum := fIntegralAccum + (_fError * tCycleTime_s / fTn_s);
END_IF

IF tCycleTime_s > 0.0001 THEN
    _fDerivative := fKp * fTv_s * ((_fError - fPreviousError) / tCycleTime_s);
ELSE
    _fDerivative := 0.0;
END_IF

fPreviousError   := _fError;
_fManipulatedVar := _fProportional + fIntegralAccum + _fDerivative;

IF _fManipulatedVar > 100.0 THEN
    _fManipulatedVar := 100.0;
ELSIF _fManipulatedVar < 0.0 THEN
    _fManipulatedVar := 0.0;
END_IF

M_ExecutePIDTuningStep := _fManipulatedVar;
END_METHOD

METHOD PUBLIC M_ExecutePneumaticValveSequence : BOOL
VAR_INPUT
    nValveIndex    : INT;
    bCommandOpen   : BOOL;
    tActuationTime : TIME;
END_VAR
VAR_OUTPUT
    bPositionConfirmed : BOOL;
    bTravelTimeout     : BOOL;
END_VAR
IF nValveIndex >= 1 AND nValveIndex <= 8 THEN
    IF bCommandOpen THEN
        bPositionConfirmed := TRUE;
        bTravelTimeout     := FALSE;
    ELSE
        bPositionConfirmed := FALSE;
        bTravelTimeout     := FALSE;
    END_IF

    M_ExecutePneumaticValveSequence := TRUE;
ELSE
    bPositionConfirmed              := FALSE;
    bTravelTimeout                  := TRUE;
    M_ExecutePneumaticValveSequence := FALSE;
END_IF
END_METHOD

METHOD PUBLIC M_FormatDiagnosticTelemetryJSON : STRING(255)
VAR_INPUT
    nBatchNum   : UDINT;
    fYield      : REAL;
    sIdentifier : STRING(80);
END_VAR
VAR
    _sOut : STRING(255);
END_VAR
_sOut := CONCAT('{"batch":', UDINT_TO_STRING(nBatchNum));
_sOut := CONCAT(_sOut, ',"id":"');
_sOut := CONCAT(_sOut, sIdentifier);
_sOut := CONCAT(_sOut, '","yield_pct":');
_sOut := CONCAT(_sOut, REAL_TO_STRING(fYield));
_sOut := CONCAT(_sOut, ',"status":"OK"}');

M_FormatDiagnosticTelemetryJSON := _sOut;
END_METHOD

METHOD PUBLIC M_PerformPreFlightSafetyAudit : BOOL
VAR_INPUT
    fMinPressure_Bar : LREAL;
    fMaxTemp_C       : REAL;
END_VAR
VAR_OUTPUT
    nAuditViolationCode : UDINT;
END_VAR
VAR
    _nIdx : INT;
END_VAR
nAuditViolationCode := 0;

FOR _nIdx := 1 TO cMaxPipelineStages DO
    IF NOT _arrNodeSnapshots[_nIdx].bActive THEN
        nAuditViolationCode := 16#A001; // Inactive node
        M_PerformPreFlightSafetyAudit := FALSE;
        RETURN;
    END_IF
END_FOR

IF fMinPressure_Bar < 0.5 THEN
    nAuditViolationCode           := 16#A002;
    M_PerformPreFlightSafetyAudit := FALSE;
    RETURN;
END_IF

M_PerformPreFlightSafetyAudit := TRUE;
END_METHOD

(*******************************************************************************
 * Method: M_ProcessSensorBatch
 * Summary: Multi-parameter (12 inputs, 3 outputs) comprehensive sensor batch
 *          evaluation and diagnostic method with deep algorithm logic.
 *******************************************************************************)
METHOD M_ProcessSensorBatch : BOOL
VAR_INPUT
    fInletFlow      : REAL;
    fOutletFlow     : REAL;
    fInletPressure  : LREAL;
    fOutletPressure : LREAL;
    fCoreTemp       : REAL;
    fJacketTemp     : REAL;
    bValveOpen      : BOOL;
    bPumpRunning    : BOOL;
    nFilterState    : INT;
    tElapsed        : TIME;
    fToleranceBand  : REAL;
    sBatchId        : STRING(80);
END_VAR
VAR_OUTPUT
    fComputedEfficiency : REAL;
    bThresholdExceeded  : BOOL;
    nAnomalyBitmask     : DWORD;
END_VAR
VAR
    _fDeltaPressure    : LREAL;
    _fTempGradient     : REAL;
    _nEvalIndex        : INT;
    _arrLocalGradients : ARRAY[1..4] OF REAL;
END_VAR
bThresholdExceeded  := FALSE;
nAnomalyBitmask     := 16#0000_0000;
fComputedEfficiency := 0.0;

{region "Sensor Delta Computation"}
    _fDeltaPressure := ABS(fInletPressure - fOutletPressure);
    _fTempGradient  := ABS(fCoreTemp - fJacketTemp);

    IF (fInletFlow > 0.0) AND (fOutletFlow >= 0.0) THEN
        fComputedEfficiency := (fOutletFlow / fInletFlow) * 100.0;

        IF fComputedEfficiency > 100.0 THEN
            fComputedEfficiency := 100.0;
    END_IF
END_IF
{endregion}

{region "Multi-Condition Anomaly Classification"}
    IF _fDeltaPressure > 2.5 THEN
        nAnomalyBitmask    := nAnomalyBitmask OR 16#0000_0001;
        bThresholdExceeded := TRUE;
END_IF

    IF _fTempGradient > 30.0 THEN
        nAnomalyBitmask    := nAnomalyBitmask OR 16#0000_0002;
        bThresholdExceeded := TRUE;
END_IF

    IF NOT bValveOpen AND bPumpRunning THEN
        nAnomalyBitmask    := nAnomalyBitmask OR 16#0000_0004;
        bThresholdExceeded := TRUE;
END_IF

    IF nFilterState < 0 THEN
        nAnomalyBitmask := nAnomalyBitmask OR 16#0000_0008;
END_IF

    IF (fToleranceBand > 0.0) AND (_fTempGradient > (50.0 * fToleranceBand)) THEN
        nAnomalyBitmask := nAnomalyBitmask OR 16#0000_0010;
END_IF
{endregion}

// Local array initialization and gradient sweep
FOR _nEvalIndex := 1 TO 4 DO
    _arrLocalGradients[_nEvalIndex] := _fTempGradient / INT_TO_REAL(_nEvalIndex);
    IF _arrLocalGradients[_nEvalIndex] > 100.0 THEN
        bThresholdExceeded := TRUE;
    END_IF
END_FOR

M_ProcessSensorBatch := (nAnomalyBitmask = 16#0000_0000) AND NOT bThresholdExceeded;
END_METHOD

METHOD PUBLIC M_RunStatisticalProcessControl : BOOL
VAR_INPUT
    arrSamples     : ARRAY[1..16] OF REAL;
    nSampleCount   : INT;
    fNominalTarget : REAL;
    fUpperLimit    : REAL;
    fLowerLimit    : REAL;
END_VAR
VAR_OUTPUT
    fCalculatedCpk : REAL;
END_VAR
VAR
    _nIdx    : INT;
    _fSum    : REAL;
    _fMean   : REAL;
    _fVarSum : REAL;
    _fSigma  : REAL;
    _fCpu    : REAL;
    _fCpl    : REAL;
    _fDiff   : REAL;
END_VAR
_fSum    := 0.0;
_fVarSum := 0.0;

IF nSampleCount <= 1 THEN
    fCalculatedCpk                 := 0.0;
    M_RunStatisticalProcessControl := FALSE;
    RETURN;
END_IF

FOR _nIdx := 1 TO nSampleCount DO
    _fSum := _fSum + arrSamples[_nIdx];
END_FOR

_fMean := _fSum / INT_TO_REAL(nSampleCount);

FOR _nIdx := 1 TO nSampleCount DO
    _fDiff   := arrSamples[_nIdx] - _fMean;
    _fVarSum := _fVarSum + (_fDiff * _fDiff);
END_FOR

_fSigma := SQRT(_fVarSum / INT_TO_REAL(nSampleCount - 1));

IF _fSigma > 0.0001 THEN
    _fCpu          := (fUpperLimit - _fMean) / (3.0 * _fSigma);
    _fCpl          := (_fMean - fLowerLimit) / (3.0 * _fSigma);
    fCalculatedCpk := MIN(_fCpu, _fCpl);
ELSE
    fCalculatedCpk := 2.0; // Perfect zero-variance process
END_IF

M_RunStatisticalProcessControl := (fCalculatedCpk >= 1.33);
END_METHOD

PROPERTY P_ActiveStage : INT
GET
P_ActiveStage := nActiveStageIndex;
END_GET
SET
IF (P_ActiveStage >= 0) AND (P_ActiveStage <= cMaxPipelineStages) THEN
    _nSubStepIndex := P_ActiveStage;
END_IF
END_SET
END_PROPERTY

PROPERTY P_IsReadyForNextBatch : BOOL
GET
P_IsReadyForNextBatch := bOperational AND NOT bProcessBusy AND NOT bFaultActive;
END_GET
END_PROPERTY

PROPERTY P_OverallHealth : REAL
GET
IF bFaultActive THEN
    P_OverallHealth := 0.0;
ELSIF bOperational THEN
    P_OverallHealth := 100.0;
ELSE
    P_OverallHealth := 50.0;
END_IF
END_GET
END_PROPERTY

PROPERTY P_ProcessStateName : STRING(80)
GET
P_ProcessStateName := sCurrentPhaseName;
END_GET
END_PROPERTY

END_FUNCTION_BLOCK

// ---- samples/FB_Sample_WidgetBase.TcPOU
FUNCTION_BLOCK FB_Sample_WidgetBase IMPLEMENTS I_Sample_WidgetInterface
VAR
    _sAdsPath : STRING(255);
    _sAttr1   : STRING(80);
    _nCalls   : UDINT;
END_VAR

;

PROPERTY AdsPath : STRING(255)
GET
AdsPath := _sAdsPath;
END_GET
END_PROPERTY

PROPERTY AttributeVariable1 : STRING(80)
GET
AttributeVariable1 := _sAttr1;
END_GET
SET
_sAttr1 := AttributeVariable1;
END_SET
END_PROPERTY

METHOD BuildAttributes : UDINT
VAR_INPUT
    nFlags : DWORD;
END_VAR
_nCalls         := _nCalls + 1;
BuildAttributes := _nCalls;
END_METHOD

METHOD ProcessCommand : BOOL
VAR_INPUT
    nCommandId : DINT;
    fValue     : LREAL;
END_VAR
VAR_OUTPUT
    bHandled : BOOL;
END_VAR
IF nCommandId = 1 THEN
    bHandled       := TRUE;
    ProcessCommand := TRUE;
ELSE
    bHandled       := FALSE;
    ProcessCommand := FALSE;
END_IF
END_METHOD

END_FUNCTION_BLOCK

// ---- syntax/F_Syntax_Add.TcPOU
FUNCTION F_Syntax_Add : INT
VAR_INPUT
    nA : INT;
    nB : INT;
END_VAR

F_Syntax_Add := nA + nB;

END_FUNCTION

// ---- syntax/F_Syntax_GenericAny.TcPOU
FUNCTION F_Syntax_GenericAny : BOOL
VAR_INPUT
    anyParam : ANY;
END_VAR
VAR
    pByte : POINTER TO BYTE;
END_VAR

IF anyParam.typeclass = __SYSTEM.TYPE_CLASS.TYPE_INT THEN
    pByte               := anyParam.pValue;
    F_Syntax_GenericAny := (pByte <> 0);
ELSE
    F_Syntax_GenericAny := FALSE;
END_IF

END_FUNCTION

// ---- syntax/F_Syntax_Return.TcPOU
FUNCTION F_Syntax_Return : BOOL
VAR_INPUT
    nValue : INT;
END_VAR

IF nValue < 0 THEN
    F_Syntax_Return := FALSE;
    RETURN;
END_IF

F_Syntax_Return := nValue > 0;

END_FUNCTION

// ---- syntax/FB_Syntax_AbstractBase.TcPOU
FUNCTION_BLOCK ABSTRACT FB_Syntax_AbstractBase IMPLEMENTS I_Syntax_Widget
VAR
    _nBaseId : DINT;
    _bReady  : BOOL;
END_VAR

METHOD ABSTRACT M_GetValue : INT
END_METHOD

METHOD M_Init : BOOL
M_Init := TRUE;
END_METHOD

METHOD ABSTRACT M_Reset : BOOL
END_METHOD

PROPERTY P_Name : STRING
GET
P_Name := 'Base';
END_GET
END_PROPERTY

PROPERTY P_Ready : BOOL
GET
P_Ready := _bReady;
END_GET
END_PROPERTY

END_FUNCTION_BLOCK

// ---- syntax/FB_Syntax_AdvancedSystemExtensions.TcPOU
FUNCTION_BLOCK FB_Syntax_AdvancedSystemExtensions IMPLEMENTS I_Syntax_BaseDevice
VAR_INPUT
    bExecute : BOOL;
    iDevice  : I_Syntax_BaseDevice;
END_VAR
VAR_OUTPUT
    bBusy  : BOOL;
    bDone  : BOOL;
    bError : BOOL;
END_VAR
VAR
    // --- 1. System Introspection & Info Types ---
    _stVarInfo     : __SYSTEM.VAR_INFO;
    _nCounter      : DINT := 100;
    _nAtomicVal    : DINT := 0;
    _nOldAtomic    : DINT;
    _dwSpinLock    : DWORD;
    _dwLockResult  : DWORD;
    _bLockAcquired : BOOL;

    // --- 2. Interface Query Pointer ---
    _pDeviceInstance : POINTER TO FB_Syntax_AdvancedSystemExtensions;
    _bPointerValid   : BOOL;

    // --- 3. Compiler Position Macros ---
    _sMacroPosition : STRING(255);
    _sMacroPOU      : STRING(80);

    // --- 4. Single FB Initializer at Declaration ---
    _fbStartupTimer : TON := (PT := T#5S);
    _fbFailsafeTon  : TON := (IN := TRUE, PT := T#2S500MS);

    // --- 5. Partial Bit / Byte / Word Access ---
    _nTestDWord : DWORD := 16#1234_5678;
    _bBitX0     : BOOL;
    _nByteB1    : BYTE;
    _nWordW1    : WORD;

    // --- 6. Pointer Indexed Access ---
    _pByteMemory : POINTER TO BYTE;
    _arrRawBytes : ARRAY[0..7] OF BYTE := [16#AA, 16#BB, 16#CC, 16#DD, 16#11, 16#22, 16#33, 16#44];
    _nExtracted  : BYTE;

    // --- 7. Fluent Builder State ---
    _fGain   : LREAL := 1.0;
    _fOffset : LREAL := 0.0;
END_VAR

// -----------------------------------------------------------------------------
// 1. System Introspection (__VARINFO)
// -----------------------------------------------------------------------------
_stVarInfo := __VARINFO(_nCounter);

// -----------------------------------------------------------------------------
// 2. Interlocked Multitask Operations (__XADD & TEST_AND_SET)
// -----------------------------------------------------------------------------
_nOldAtomic    := __XADD(ADR(_nAtomicVal), 1);
_dwLockResult  := TEST_AND_SET(_dwSpinLock);
_bLockAcquired := (_dwLockResult = 1);

// -----------------------------------------------------------------------------
// 3. Compiler Position Macros
// -----------------------------------------------------------------------------
_sMacroPosition := __POSITION();
_sMacroPOU      := __POUNAME();

// -----------------------------------------------------------------------------
// 4. Interface to Pointer Dynamic Resolution (__QUERYPOINTER)
// -----------------------------------------------------------------------------
IF iDevice <> 0 THEN
    _bPointerValid := __QUERYPOINTER(iDevice, _pDeviceInstance);
END_IF

// -----------------------------------------------------------------------------
// 5. Partial Variable Bit / Byte / Word Access (%X, %B, %W, %D)
// -----------------------------------------------------------------------------
_bBitX0  := _nTestDWord.%X0;
_nByteB1 := _nTestDWord.%B1;
_nWordW1 := _nTestDWord.%W1;

_nTestDWord.%X31 := TRUE;
_nTestDWord.%B0  := 16#FF;

// -----------------------------------------------------------------------------
// 6. Pointer Array Index Access
// -----------------------------------------------------------------------------
_pByteMemory := ADR(_arrRawBytes[0]);

IF _pByteMemory <> 0 THEN
    _nExtracted     := _pByteMemory[2];
    _pByteMemory[3] := 16#EE;
END_IF

// -----------------------------------------------------------------------------
// 7. Generic ANY Parameter Call
// -----------------------------------------------------------------------------
F_Syntax_GenericAny(anyParam := _nCounter);
F_Syntax_GenericAny(anyParam := _arrRawBytes);

// -----------------------------------------------------------------------------
// 8. Method Chaining (Fluent Interface Pattern)
// -----------------------------------------------------------------------------
THIS^.M_SetGain(2.5).M_SetOffset(10.0);

// -----------------------------------------------------------------------------
// 9. Single FB Execution
// -----------------------------------------------------------------------------
_fbStartupTimer(IN := bExecute);
bDone := _fbStartupTimer.Q;

METHOD M_Reset : BOOL
_nCounter := 0;
M_Reset   := TRUE;
END_METHOD

METHOD M_SetGain : REFERENCE TO FB_Syntax_AdvancedSystemExtensions
VAR_INPUT
    fGain : LREAL;
END_VAR
_fGain := fGain;
M_SetGain REF= THIS^;
END_METHOD

METHOD M_SetOffset : REFERENCE TO FB_Syntax_AdvancedSystemExtensions
VAR_INPUT
    fOffset : LREAL;
END_VAR
_fOffset := fOffset;
M_SetOffset REF= THIS^;
END_METHOD

METHOD M_Start : BOOL
VAR_INPUT
    bForce : BOOL;
END_VAR
bBusy   := TRUE;
M_Start := TRUE;
END_METHOD

METHOD M_Stop : BOOL
bBusy  := FALSE;
M_Stop := TRUE;
END_METHOD

PROPERTY P_IsRunning : BOOL
GET
P_IsRunning := bBusy;
END_GET
END_PROPERTY

END_FUNCTION_BLOCK

// ---- syntax/FB_Syntax_AssignAlignmentHeuristics.TcPOU
FUNCTION_BLOCK FB_Syntax_AssignAlignmentHeuristics
VAR
    stDeviceControl                   : ST_Syntax_Mini;
    bCmdA                             : BOOL;
    bCmdB                             : BOOL;
    bCmdC                             : BOOL;
    nShort                            : INT;
    nVeryLongVariableNameForAlignment : DINT;
    nOther                            : DINT;
    nIdx                              : INT;
END_VAR

// 1. Chained assignments
bCmdA := bCmdB := FALSE;
bCmdA := bCmdB := TRUE;

// 2. 3-line qualified assignment group with same base variable
stDeviceControl.nId     := 10;
stDeviceControl.bActive := TRUE;
stDeviceControl.sName   := 'DeviceMain';

// 3. Simple assignment group alignment
nShort                            := 1;
nVeryLongVariableNameForAlignment := 200;
nOther                            := 3;

// 4. FOR-loop assignment alignment
FOR nIdx := 1 TO 5 DO
    stDeviceControl.nId     := nIdx;
    stDeviceControl.bActive := FALSE;
END_FOR

END_FUNCTION_BLOCK

// ---- syntax/FB_Syntax_AttributesComprehensive.TcPOU
// 1. Multiple attributes on POU level (stacked)
{attribute 'reflection'}
{attribute 'hide_all_locals'}
{attribute 'no_explicit_call' := 'Call methods instead of FB body directly'}
FUNCTION_BLOCK FB_Syntax_AttributesComprehensive
VAR_INPUT
    // 2. Attribute above variable (standard single line)
    {attribute 'TcEncoding' := 'UTF-8'}
    sUtf8Input : STRING(255);

    // 3. Attribute inline before variable name
    {attribute 'hide'} bHiddenFlag : BOOL;

    // Normal input for alignment reference
    nNormalInput : INT := 10;
END_VAR
VAR_OUTPUT
    // 4. Attribute with value without spaces around :=
    {attribute 'displaymode':='hex'}
    dwStatusHex : DWORD;

    // Normal output
    bDone : BOOL;
END_VAR
VAR
    // 5. Multiple stacked attributes above a variable
    {attribute 'reflection'}
    {attribute 'instance-path'}
    {attribute 'noinit'}
    _sInstancePath : STRING(255);

    // 6. Multiple inline attributes on one line before variable
    {attribute 'hide'} {attribute 'noinit'} _nInternalCached : DINT;

    // 7. Attribute above variable with initial assignment and inline comment
    {attribute 'TcLinkTo' := 'TIID^Device 1^Term 1^Channel 1^Input'}
    _bHardwareInput : BOOL := FALSE; (* Linked to EtherCAT terminal *)

    _nCycleCount : UDINT;
END_VAR

// Increment cycle
_nCycleCount := _nCycleCount + 1;
bDone        := TRUE;
dwStatusHex  := 16#A5A5;

// 8. Attribute on method level
{attribute 'TcRpcEnable'}
METHOD M_ProtectedAction : BOOL
VAR_INPUT
    {attribute 'hide'}
    nSecretCode : INT;
END_VAR
M_ProtectedAction := (nSecretCode = 42);
END_METHOD

// 9. Attribute on property level
{attribute 'monitoring' := 'call'}
PROPERTY P_Diagnostics : STRING
GET
P_Diagnostics := _sInstancePath;
END_GET
END_PROPERTY

END_FUNCTION_BLOCK

// ---- syntax/FB_Syntax_BitAccess.TcPOU
FUNCTION_BLOCK FB_Syntax_BitAccess
VAR
    nRegister : WORD;
    nFlags    : BYTE;
    bState    : BOOL;
    stBits    : ST_Syntax_Bitfields;
END_VAR

nRegister.0  := TRUE;
nRegister.15 := FALSE;
bState       := nRegister.7;

nFlags.0 := bState;
nFlags.1 := NOT stBits.bBit0;

stBits.bBit0 := TRUE;
stBits.bBit1 := FALSE;
stBits.bBit2 := nFlags.2;

END_FUNCTION_BLOCK

// ---- syntax/FB_Syntax_CaseRanges.TcPOU
FUNCTION_BLOCK FB_Syntax_CaseRanges
VAR_INPUT
    nSelector : INT;
    nSub      : INT;
END_VAR
VAR
    nResult : INT;
END_VAR

CASE nSelector OF
    1, 2, 3:
        nResult := 10;
    4..7:
        CASE nSub OF
            0:
                nResult := 20;
            1..3:
                nResult := 30;
        ELSE
            nResult := -1;
        END_CASE
    8..10, 15:
        nResult := 40;
ELSE
    nResult := 0;
END_CASE

END_FUNCTION_BLOCK

// ---- syntax/FB_Syntax_ComplexExpressions.TcPOU
FUNCTION_BLOCK FB_Syntax_ComplexExpressions
VAR
    bA       : BOOL;
    bB       : BOOL;
    bC       : BOOL;
    bD       : BOOL;
    bResult  : BOOL;
    fVal1    : LREAL := 3.14159;
    fVal2    : LREAL := 2.71828;
    fVal3    : LREAL := 1.41421;
    fOut     : LREAL;
    nIndex   : INT                 := 2;
    arrData  : ARRAY[0..9] OF DINT := [0, 10, 20, 30, 40, 50, 60, 70, 80, 90];
    pData    : POINTER TO DINT;
    dwMask   : DWORD := 16#FF00AA55;
    dwResult : DWORD;
END_VAR

// 1. Chained boolean operators with ExST short-circuiting
bResult := (bA AND_THEN bB) OR_ELSE (bC AND NOT bD) OR (bA XOR bC);

// 2. Nested mathematical function calls and precedence
fOut := LIMIT(0.0, SQRT(ABS(SIN(fVal1) * COS(fVal2) + EXPT(fVal3, 2.0))), 100.0);

// 3. Selection operators (SEL, MUX, MIN, MAX)
fOut := SEL(bResult, MIN(fVal1, fVal2), MAX(fVal2, fVal3));
fOut := MUX(
        nIndex,
        0.0,
        fVal1,
        fVal2,
        fVal3,
        99.9);

// 4. Bitwise shifts and mask operations
dwResult := (SHL(dwMask, 4) OR SHR(dwMask, 2)) AND 16#FFFF0000 XOR 16#0000FFFF;

// 5. Pointers and address resolution
pData := ADR(arrData[nIndex]);

IF pData <> 0 THEN
    pData^ := pData^ + 1;
END_IF

END_FUNCTION_BLOCK

// ---- syntax/FB_Syntax_ComplexInits.TcPOU
FUNCTION_BLOCK FB_Syntax_ComplexInits
VAR
    stConfig : ST_Syntax_Mini                := (nId := 10, bActive := TRUE, sName := 'InitTag');
    aNumbers : ARRAY[1..5] OF INT            := [10, 20, 30, 40, 50];
    aStructs : ARRAY[1..2] OF ST_Syntax_Mini := [(nId := 1, bActive := FALSE, sName := 'First'), (nId := 2, bActive := TRUE, sName := 'Second')];
    a2D      : ARRAY[1..2, 1..2] OF INT      := [1, 2, 3, 4];
END_VAR

IF stConfig.nId = 10 THEN
    stConfig.nId     := 20;
    stConfig.bActive := FALSE;
    stConfig.sName   := 'UpdatedTag';
END_IF

END_FUNCTION_BLOCK

// ---- syntax/FB_Syntax_DeepNesting.TcPOU
FUNCTION_BLOCK FB_Syntax_DeepNesting
VAR
    nOuter : INT;
    nInner : INT;
    nDeep  : INT;
    bFlag1 : BOOL;
    bFlag2 : BOOL;
    bFlag3 : BOOL;
    nTotal : DINT;
END_VAR

IF bFlag1 THEN
    FOR nOuter := 1 TO 5 DO
        IF bFlag2 THEN
            CASE nOuter OF
                1:
                    WHILE nInner < 3 DO
                        IF bFlag3 THEN
                            REPEAT
                                nDeep  := nDeep + 1;
                                nTotal := nTotal + (nOuter * nInner * nDeep);
                            UNTIL nDeep >= 5
                            END_REPEAT;
                        ELSE
                            nTotal := nTotal + 1;
                        END_IF

                        nInner := nInner + 1;
                    END_WHILE
                2..4:
                    nTotal := nTotal + 10;
            ELSE
                nTotal := 0;
            END_CASE
        END_IF
    END_FOR
END_IF

END_FUNCTION_BLOCK

// ---- syntax/FB_Syntax_Derived.TcPOU
FUNCTION_BLOCK FB_Syntax_Derived EXTENDS FB_Syntax_AbstractBase IMPLEMENTS I_Syntax_Extended
VAR
    _sStatus  : STRING := 'IDLE';
    _nCounter : DINT;
END_VAR

_nCounter := _nCounter + 1;

METHOD M_Execute : BOOL
VAR_INPUT
    nCommand : DINT;
END_VAR
CASE nCommand OF
    1:
        _sStatus := 'RUNNING';
    2:
        _sStatus := 'PAUSED';
ELSE
    _sStatus := 'UNKNOWN';
END_CASE
M_Execute := TRUE;
END_METHOD

METHOD M_GetValue : INT
M_GetValue := TO_INT(_nCounter);
END_METHOD

METHOD M_Reset : BOOL
_nCounter := 0;
_bReady   := TRUE;
_sStatus  := 'RESET';
M_Reset   := TRUE;
END_METHOD

PROPERTY P_ExtendedStatus : INT
GET
P_ExtendedStatus := 1;
END_GET
END_PROPERTY

PROPERTY P_Status : STRING
GET
P_Status := _sStatus;
END_GET
END_PROPERTY

END_FUNCTION_BLOCK

// ---- syntax/FB_Syntax_DynamicMem.TcPOU
FUNCTION_BLOCK FB_Syntax_DynamicMem
VAR
    pDyn    : POINTER TO ST_Syntax_Dyn;
    bNew    : BOOL := TRUE;
    bDelete : BOOL;
END_VAR

IF bNew AND (pDyn = 0) THEN
    pDyn := __NEW(ST_Syntax_Dyn);
    bNew := FALSE;
END_IF

IF bDelete THEN
    __DELETE(pDyn);
    bDelete := FALSE;
END_IF

END_FUNCTION_BLOCK

// ---- syntax/FB_Syntax_ExhaustiveComments.TcPOU
(*******************************************************************************
 * POU Name:    FB_Syntax_ExhaustiveComments
 * Description: Comprehensive test fixture for ALL TwinCAT 3 IEC 61131-3
 *              comment variants (line //, block (* *), nested, inline).
*******************************************************************************)
FUNCTION_BLOCK FB_Syntax_ExhaustiveComments
VAR_INPUT (* Inputs section *)
    /// <summary>Enable command</summary>
    bEnable : BOOL := FALSE; (* Master enable flag *)
    nSetVal : INT  := 100;   // Target value setpoint
    fLimit  : REAL := 99.5;  (* Upper threshold in [degC] *)
END_VAR
VAR_OUTPUT (* Outputs section *)
    /// <summary>Active status</summary>
    bActive     : BOOL;  (* Currently operational *)
    bError      : BOOL;  // Error indicator
    nStatusCode : UDINT; (* Diagnostic code: 16#0000_0000 = OK *)
END_VAR
VAR_IN_OUT (* In-Out variables *)
    stGlobalCtx : ST_Syntax_Mini; (* Shared context structure *)
END_VAR
VAR (* Internal state variables *)
    // --- 1. Control flags ---
    _bInitDone : BOOL := FALSE; (* First-cycle init marker *)
    _nCycleCnt : UDINT;         // Total executed cycles

    // --- 2. State machine ---
    _nStep    : INT := 0; (* Current step index *)
    _nSubStep : INT := 0; // Secondary step

    // --- 3. Arithmetic values ---
    _fAccum     : LREAL := 0.0; (* Filtered accumulator *)
    _fbTonDelay : TON;          (* Failsafe timer *)

    (*
     * Multi-line block comment inside declaration block
     * Explaining temporary calculation buffers
     *)
    _arrScratch : ARRAY[1..4] OF DINT := [
        10, (* buffer 1 *)
        20, (* buffer 2 *)
        30, (* buffer 3 *)
        40  (* buffer 4 *)
    ];
END_VAR
VAR_TEMP (* Temporary cycle-local variables *)
    _nTempLoop  : INT;  // Loop counter
    _bCondition : BOOL; (* Transient flag *)
END_VAR

// =============================================================================
// 1. NESTED BLOCK COMMENTS & DOC COMMENTS
// =============================================================================
(* Outer comment level 1
   (* Nested comment level 2
      (* Deep nested comment level 3: x := 5; IF y THEN z := 1; END_IF; *)
Back TO level 2
*)
Back TO level 1
*)

/// Triple slash documentation comment
// Standard line comment with special chars: <XML attr="val"> & 'quotes' "double"

// =============================================================================
// 2. COMMENTS INSIDE ARITHMETIC & BOOLEAN EXPRESSIONS
// =============================================================================
_fAccum := _fAccum + (* term 1 *) (LREAL#1.5 * (* term 2 *) DINT_TO_LREAL(nSetVal)) - (* term 3 *) (fLimit / (* term 4 *) 2.0);

_bCondition := (bEnable (* check enable *) AND NOT bError (* check error *)) OR_ELSE (* fallback check *) (_nStep = 999 (* emergency *));

// =============================================================================
// 3. COMMENTS IN IF / ELSIF / ELSE CONTROL FLOW
// =============================================================================
IF (* condition check *) _bCondition THEN // branch 1 taken
    // Internal comment
    _nStep := 10; (* move to running step *)
ELSIF (* alternate check *) bError THEN (* branch error *)
    _nStep := 99; // error recovery step
ELSE (* default fallback *)
    _nStep := 0;  (* stay in idle *)
END_IF
(* end of state check *)
;

// =============================================================================
// 4. COMMENTS IN CASE STATEMENT
// =============================================================================
CASE (* evaluate active step *) _nStep OF
    0 (* Step: Idle *):
        // Idle actions
        IF bEnable THEN
            _nStep := 10; // start cycle
        END_IF

    10 (* Step: Running *), 20 (* Step: Processing *):
        // Active processing
        _nCycleCnt := _nCycleCnt + 1; (* increment cycle *)

    99 (* Step: Error *):
        // Error handling
        bError := TRUE;

ELSE (* Step: Unhandled *)
    _nStep := 0; // return to idle
END_CASE
(* end of case evaluation *)
;

// =============================================================================
// 5. COMMENTS IN LOOPS (FOR, WHILE, REPEAT)
// =============================================================================
FOR _nTempLoop := 1 (* start *) TO 4 (* stop *) BY 1 (* step *) DO
    // Array element update
    _arrScratch[_nTempLoop] := _arrScratch[_nTempLoop] + (* offset *) 1;
    IF _arrScratch[_nTempLoop] > 100 THEN
        CONTINUE; // skip rest of loop
    END_IF
END_FOR
(* end of for loop *)
;

WHILE (* guard condition *) (_nSubStep < 5) AND NOT bError DO
    _nSubStep := _nSubStep + 1; // advance sub-step
    IF _nSubStep >= 3 THEN
        EXIT; (* break early *)
    END_IF
END_WHILE
(* end of while loop *)
;

REPEAT
    _nSubStep := _nSubStep - 1; // decrement
UNTIL (* termination condition *) (_nSubStep <= 0)
END_REPEAT
(* end of repeat loop *)
;

// =============================================================================
// 6. COMMENTS IN FB CALLS & FUNCTION CALLS
// =============================================================================
_fbTonDelay(
        IN := (* trigger signal *) (bEnable AND NOT bError), // enable
        PT := (* duration *) T#500MS                        (* 500 ms delay *)
        ); // timer instance call

bActive := _fbTonDelay.Q; // output assignment

(*******************************************************************************
 * Method: M_DiagnosticReport
 * Summary: Generates diagnostic string with nested comments.
 *******************************************************************************)
METHOD M_DiagnosticReport : STRING(255)
VAR_INPUT
    nDetailLevel : INT; (* 0=brief, 1=full *)
END_VAR
VAR
    sReport : STRING(255); // Output accumulator
END_VAR
// Build report string
IF nDetailLevel > 0 THEN
    (* Full detail formatting *)
    sReport := CONCAT((* prefix *) 'Status: ', (* value *) UDINT_TO_STRING(nStatusCode) );
ELSE
    (* Brief formatting *)
    sReport := 'OK';
END_IF

M_DiagnosticReport := sReport; // Return result
END_METHOD

PROPERTY P_IsReady : BOOL
GET
// Getter logic
P_IsReady := _bInitDone AND NOT bError; (* Ready when initialized and no error *)
END_GET
END_PROPERTY

// ---- syntax/FB_Syntax_ExST.TcPOU
FUNCTION_BLOCK FB_Syntax_ExST
VAR
    nI      : INT;
    nSum    : INT;
    bFlag   : BOOL;
    rRef    : REFERENCE TO INT;
    nTarget : INT;
END_VAR

IF (nI <> 0) AND_THEN (nSum > 0) OR bFlag THEN
    nSum := nSum + 1;
END_IF

FOR nI := 1 TO 5 DO
    IF nI MOD 2 = 0 THEN
        CONTINUE;
    END_IF

    nSum := nSum + nI;
END_FOR

JMP _skip;
nSum := -1;
_skip:

rRef REF= nTarget;
rRef := 42;

END_FUNCTION_BLOCK

// ---- syntax/FB_Syntax_FBInitMethods.TcPOU
FUNCTION_BLOCK FB_Syntax_FBInitMethods
VAR
    _nId       : DINT;
    _sLabel    : STRING(80);
    _bInitDone : BOOL;
END_VAR

METHOD FB_exit : BOOL
VAR_INPUT
    bInCopyCode : BOOL; // if TRUE, the exit method is called for exiting an instance that is copied afterwards (online change).
END_VAR
_bInitDone := FALSE;
FB_exit    := TRUE;
END_METHOD

METHOD FB_init : BOOL
VAR_INPUT
    bInitRetains : BOOL; // if TRUE, the retain variables are initialized (warm start / cold start)
    bInCopyCode  : BOOL; // if TRUE, the instance afterwards gets moved into the copy code (online change)
    nInitialId   : DINT;
    sInitialName : STRING(80);
END_VAR
_nId       := nInitialId;
_sLabel    := sInitialName;
_bInitDone := TRUE;
FB_init    := TRUE;
END_METHOD

METHOD FB_reinit : BOOL
_bInitDone := TRUE;
FB_reinit  := TRUE;
END_METHOD

END_FUNCTION_BLOCK

// ---- syntax/FB_Syntax_IfMultilineCalls.TcPOU
FUNCTION_BLOCK FB_Syntax_IfMultilineCalls
VAR
    sStr1   : STRING(80);
    sStr2   : STRING(80);
    sResult : STRING(255);
    rTarget : REFERENCE TO INT;
    nVal    : INT;
    bOk     : BOOL;
END_VAR

IF len(sStr1) > 0 AND len(sStr2) > 0 THEN
    bOk := FALSE;
ELSE
    bOk := TRUE;
END_IF

IF NOT __ISVALIDREF(rTarget) THEN
    nVal := 0;
ELSE
    nVal := rTarget;
END_IF

IF (len(sStr1) > 0) AND (len(sStr2) > 0) AND (len(sResult) = 0) THEN
    bOk := TRUE;
END_IF

END_FUNCTION_BLOCK

// ---- syntax/FB_Syntax_LargeServicePOU.TcPOU
FUNCTION_BLOCK FB_Syntax_LargeServicePOU
VAR_INPUT
    bEnable    : BOOL;
    tCycleTime : TIME := T#10MS;
END_VAR
VAR_OUTPUT
    bActive     : BOOL;
    bError      : BOOL;
    hrErrorCode : HRESULT;
    sStatusMsg  : STRING(255);
END_VAR
VAR
    _nState       : INT;
    _nCount       : DINT;
    _fThroughput  : LREAL;
    _nMaxRetries  : UINT := 3;
    _stTreeConfig : ST_Syntax_ComplexTree;
    _fbTimer      : TON;
END_VAR

IF NOT bEnable THEN
    _nState := 0;
    bActive := FALSE;
    RETURN;
END_IF

bActive := TRUE;
_fbTimer(IN := (_nState > 0), PT := tCycleTime);

CASE _nState OF
    0:
        IF THIS^.M_Initialize(bForce := FALSE) THEN
            _nState := 10;
        END_IF

    10:
        _nCount := _nCount + 1;
        IF _fbTimer.Q THEN
            A_UpdateStats();
            _nState := 20;
        END_IF

    20:
        IF THIS^.P_IsBusy THEN
            ;
        ELSE
            _nState := 10;
        END_IF

    99:
        A_HandleErrors();
END_CASE

ACTION A_HandleErrors:
bError      := TRUE;
hrErrorCode := 16#80004005;
sStatusMsg  := 'Service encountered an unrecoverable fault';
END_ACTION

ACTION A_UpdateStats:
_fThroughput := DINT_TO_LREAL(_nCount) / 10.0;
END_ACTION

METHOD M_Configure : BOOL
VAR_INPUT
    stConfig : ST_Syntax_ComplexTree;
END_VAR
_stTreeConfig := stConfig;
M_Configure   := TRUE;
END_METHOD

METHOD M_Execute : HRESULT
VAR_INPUT
    fInput : LREAL;
END_VAR
VAR_OUTPUT
    fResult  : LREAL;
    bSuccess : BOOL;
END_VAR
IF fInput < 0.0 THEN
    fResult   := 0.0;
    bSuccess  := FALSE;
    M_Execute := 16#80070057; // E_INVALIDARG
    RETURN;
END_IF

fResult   := SQRT(fInput) * 2.5;
bSuccess  := TRUE;
M_Execute := 0; // S_OK
END_METHOD

METHOD M_Initialize : BOOL
VAR_INPUT
    bForce : BOOL;
END_VAR
IF bForce OR (_nState = 0) THEN
    _nCount      := 0;
    _fThroughput := 0.0;
    bError       := FALSE;
    hrErrorCode  := 0;
    sStatusMsg   := 'Initialized';
    M_Initialize := TRUE;
ELSE
    M_Initialize := FALSE;
END_IF
END_METHOD

METHOD M_ProcessBatch : DINT
VAR_INPUT
    arrData : ARRAY[1..10] OF LREAL;
END_VAR
VAR
    i      : INT;
    nValid : DINT;
END_VAR
nValid := 0;

FOR i := 1 TO 10 DO
    IF arrData[i] > 0.0 THEN
        nValid := nValid + 1;
    END_IF
END_FOR

M_ProcessBatch := nValid;
END_METHOD

METHOD M_Reset : BOOL
_nState := 0;
bError  := FALSE;
M_Reset := TRUE;
END_METHOD

PROPERTY P_CurrentThroughput : LREAL
GET
P_CurrentThroughput := _fThroughput;
END_GET
END_PROPERTY

PROPERTY P_IsBusy : BOOL
GET
P_IsBusy := (_nState >= 10) AND (_nState < 90);
END_GET
END_PROPERTY

PROPERTY P_MaxRetries : UINT
GET
P_MaxRetries := _nMaxRetries;
END_GET
SET
IF P_MaxRetries > 0 AND P_MaxRetries <= 10 THEN
    _nMaxRetries := P_MaxRetries;
END_IF
END_SET
END_PROPERTY

END_FUNCTION_BLOCK

// ---- syntax/FB_Syntax_LoopControl.TcPOU
FUNCTION_BLOCK FB_Syntax_LoopControl
VAR
    nSum       : DINT;
    nCountdown : INT;
    nStepState : INT;
    bFound     : BOOL;
    arrBuffer  : ARRAY[1..10] OF INT;
END_VAR

nSum := 0;

// FOR loop forward
FOR nCountdown := 1 TO 10 DO
    arrBuffer[nCountdown] := nCountdown * 2;
    nSum                  := nSum + arrBuffer[nCountdown];
END_FOR

// FOR loop backwards with step
FOR nCountdown := 10 TO 1 BY -2 DO
    IF arrBuffer[nCountdown] > 10 THEN
        CONTINUE;
    END_IF

    nSum := nSum - arrBuffer[nCountdown];
END_FOR

// WHILE loop with EXIT
nCountdown := 1;

WHILE nCountdown <= 10 DO
    IF arrBuffer[nCountdown] = 6 THEN
        bFound := TRUE;
        EXIT;
    END_IF

    nCountdown := nCountdown + 1;
END_WHILE

// REPEAT UNTIL loop
nCountdown := 5;

REPEAT
    nCountdown := nCountdown - 1;
UNTIL nCountdown <= 0
END_REPEAT

// CASE with ranges and comma lists
CASE nStepState OF
    0:
        nSum := 0;
    1..5:
        nSum := nSum + 10;
    6, 7, 8:
        nSum := nSum + 20;
    9..15, 20..25:
        nSum := nSum + 50;
ELSE
    nSum := -1;
END_CASE

END_FUNCTION_BLOCK

// ---- syntax/FB_Syntax_MathOperators.TcPOU
FUNCTION_BLOCK FB_Syntax_MathOperators
VAR
    fInA, fInB, fResult : LREAL;
    nInA, nInB, nResult : DINT;
    wInA, wResult       : WORD;
    bSelect             : BOOL;
    nSelectIndex        : INT;
END_VAR

// Numeric functions
fResult := ABS(fInA);
fResult := SQRT(fInA);
fResult := LN(fInA);
fResult := LOG(fInA);
fResult := EXP(fInA);
fResult := SIN(fInA);
fResult := COS(fInA);
fResult := TAN(fInA);
fResult := ASIN(fInA);
fResult := ACOS(fInA);
fResult := ATAN(fInA);
fResult := EXPT(fInA, 2.0);

// Selection and limiting
fResult := LIMIT(0.0, fInA, 100.0);
fResult := MIN(fInA, fInB);
fResult := MAX(fInA, fInB);
fResult := SEL(bSelect, fInA, fInB);
nResult := MUX(
        nSelectIndex,
        10,
        20,
        30,
        40);

// Bit shift and rotate
wResult := SHL(wInA, 2);
wResult := SHR(wInA, 2);
wResult := ROL(wInA, 1);
wResult := ROR(wInA, 1);

END_FUNCTION_BLOCK

// ---- syntax/FB_Syntax_MultiDimArraysAndInits.TcPOU
FUNCTION_BLOCK FB_Syntax_MultiDimArraysAndInits
VAR
    arr2D       : ARRAY[1..3, 1..4] OF INT;
    arr3D       : ARRAY[0..1, 0..1, 0..1] OF BOOL;
    arrFlatInit : ARRAY[1..12] OF INT := [
        1, 2, 3, 4,
        5, 6, 7, 8,
        9, 10, 11, 12
    ];
    arrTreeNodes : ARRAY[1..2] OF ST_Syntax_ComplexTree := [
        (
            nNodeId         := 100,
            sNodeName       := 'PrimaryNode',
            eState          := E_Syntax_ExplicitIntTyped.Running,
            arrCoefficients := [1.1, 2.2, 3.3, 4.4, 5.5],
            bActive         := TRUE,
            tLastUpdated    := T#1S
        ),
        (
            nNodeId         := 200,
            sNodeName       := 'SecondaryNode',
            eState          := E_Syntax_ExplicitIntTyped.Init,
            arrCoefficients := [0.1, 0.2, 0.3, 0.4, 0.5],
            bActive         := FALSE,
            tLastUpdated    := T#500MS
        )
    ];
END_VAR

arr2D[1, 1]             := arr2D[2, 2] + arr2D[3, 3];
arr3D[0, 1, 0]          := NOT arr3D[1, 0, 1];
arrTreeNodes[1].bActive := TRUE;

END_FUNCTION_BLOCK

// ---- syntax/FB_Syntax_NestedLogCall.TcPOU
FUNCTION_BLOCK FB_Syntax_NestedLogCall
VAR
    _sPath         : STRING(255);
    _fbChild       : FB_Syntax_Calls;
    _tValue        : TIME := T#2S500MS;
    _sLog          : STRING(255);
    _sNested10     : STRING(255);
    _sReport       : STRING(255);
    _sFormatted    : STRING(255);
    _nResult       : INT;
    _nNestedMath10 : INT;
    _nIndex        : INT := 1;
    _fRealResult   : REAL;
    _arrData       : ARRAY[1..10] OF INT;
    _bCondition    : BOOL;
END_VAR

// -----------------------------------------------------------------------------
// 1. Original 3-level CONCAT log call within nested IF
// -----------------------------------------------------------------------------
IF TRUE THEN
    IF FALSE THEN
        ;
    ELSE
        _sLog := CONCAT('_fbChild: ', CONCAT(INT_TO_STRING(_fbChild.stParam.nId), CONCAT(' Value: ', INT_TO_STRING(_fbChild.nResult))));
    END_IF
END_IF

// -----------------------------------------------------------------------------
// 2. Deeply nested 10-level CONCAT string call
// -----------------------------------------------------------------------------
_sNested10 := CONCAT('1:', CONCAT('2:', CONCAT('3:', CONCAT('4:', CONCAT('5:', CONCAT('6:', CONCAT('7:', CONCAT('8:', CONCAT('9:', '10')))))))));

// -----------------------------------------------------------------------------
// 3. Deeply nested 10-level arithmetic / function call chain
// -----------------------------------------------------------------------------
_nNestedMath10 := F_Syntax_Add(1, F_Syntax_Add(2, F_Syntax_Add(3, F_Syntax_Add(4, F_Syntax_Add(5, F_Syntax_Add(6, F_Syntax_Add(7, F_Syntax_Add(8, F_Syntax_Add(9, 10)))))))));

// -----------------------------------------------------------------------------
// 4. Nested math pipeline with standard functions: MAX, MIN, LIMIT, ABS, SQRT
// -----------------------------------------------------------------------------
_nResult := MAX(0, MIN(1000, LIMIT(10, ABS(F_Syntax_Add(F_Syntax_Add(10, 20), F_Syntax_Add(30, F_Syntax_Add(40, 50)))), 500)));

_fRealResult := SQRT(INT_TO_REAL(MAX(1, MIN(100, F_Syntax_Add(F_Syntax_Add(1, 2), F_Syntax_Add(3, F_Syntax_Add(4, 5)))))));

// -----------------------------------------------------------------------------
// 5. Nested MUX and SEL calls with nested arguments
// -----------------------------------------------------------------------------
_nResult := MUX(_nIndex, F_Syntax_Add(1, 1), SEL(_bCondition, F_Syntax_Add(2, F_Syntax_Add(3, 4)), F_Syntax_Add(5, F_Syntax_Add(6, F_Syntax_Add(7, 8)))), F_Syntax_Add(9, 10));

// -----------------------------------------------------------------------------
// 6. Nested Named Parameter calls (nA := ..., nB := ...)
// -----------------------------------------------------------------------------
_nResult := F_Syntax_Add(nA := F_Syntax_Add(nA := F_Syntax_Add(nA := 1, nB := 2), nB := 3), nB := F_Syntax_Add(nA := 4, nB := F_Syntax_Add(nA := 5, nB := 6)));

// -----------------------------------------------------------------------------
// 7. Nested Calls as Array Index Expressions and Assignments
// -----------------------------------------------------------------------------
_arrData[F_Syntax_Add(1, F_Syntax_Add(0, 1))] := F_Syntax_Add(F_Syntax_Add(1, 2), F_Syntax_Add(3, F_Syntax_Add(4, 5)));

// -----------------------------------------------------------------------------
// 8. Nested Calls inside Control Flow Conditionals (IF, CASE, WHILE)
// -----------------------------------------------------------------------------
IF (F_Syntax_Add(F_Syntax_Add(1, 2), F_Syntax_Add(3, 4)) > 5) AND (F_Syntax_Add(5, F_Syntax_Add(6, 7)) < 100) THEN
    _bCondition := TRUE;
ELSIF (F_Syntax_Add(1, F_Syntax_Add(2, F_Syntax_Add(3, 4))) = 10) THEN
    _bCondition := FALSE;
END_IF

// -----------------------------------------------------------------------------
// 9. 10-level nested Boolean negation and type conversions
// -----------------------------------------------------------------------------
_bCondition := NOT (NOT (NOT (NOT (NOT (NOT (NOT (NOT (NOT (F_Syntax_Add(1, 2) = 3)))))))));
_sFormatted := TO_STRING(TO_DINT(TO_REAL(TO_INT(TO_BYTE(TO_WORD(TO_DWORD(TO_UDINT(TO_LREAL(F_Syntax_Add(10, 20))))))))));

// -----------------------------------------------------------------------------
// 10. 10-level nested MIN/MAX chain and 10-level nested parentheses arithmetic
// -----------------------------------------------------------------------------
_nResult := MIN(100, MIN(90, MIN(80, MIN(70, MIN(60, MIN(50, MIN(40, MIN(30, MIN(20, MAX(1, 10))))))))));
_nResult := (1 + (2 * (3 + (4 * (5 + (6 * (7 + (8 * (9 + F_Syntax_Add(1, 2))))))))));

// -----------------------------------------------------------------------------
// 11. Multi-parameter 5-argument function calls with nested arguments
// -----------------------------------------------------------------------------
_nResult := F_5Args(
        a := F_Syntax_Add(1, 2),
        b := F_Syntax_Add(3, 4),
        c := F_Syntax_Add(5, 6),
        d := F_Syntax_Add(7, 8),
        e := F_Syntax_Add(9, 10));

// -----------------------------------------------------------------------------
// 12. Nested Logging / String Conversion Formatting
// -----------------------------------------------------------------------------
_sReport := CONCAT('Prefix: ', CONCAT(INT_TO_STRING(_fbChild.stParam.nId), CONCAT(' | Result: ', CONCAT(INT_TO_STRING(F_Syntax_Add(F_Syntax_Add(1, 2), F_Syntax_Add(3, 4))), CONCAT(' | Time: ', TO_STRING(_tValue))))));

END_FUNCTION_BLOCK

// ---- syntax/FB_Syntax_OOP.TcPOU
FUNCTION_BLOCK FB_Syntax_OOP
VAR
    _nInternal : INT;
END_VAR

_nInternal := _nInternal + 1;

METHOD M_Increment : BOOL
VAR_INPUT
    nDelta : INT;
END_VAR
_nInternal  := _nInternal + nDelta;
M_Increment := TRUE;
END_METHOD

PROPERTY P_Count : INT
GET
P_Count := _nInternal;
END_GET
END_PROPERTY

END_FUNCTION_BLOCK

// ---- syntax/FB_Syntax_Pragmas.TcPOU
FUNCTION_BLOCK FB_Syntax_Pragmas
VAR
    nValue : INT;
END_VAR

{region 'Init'}
    nValue := 1;
{endregion}

{formatting.disable}
nValue := 99;
{formatting.enable}

END_FUNCTION_BLOCK

// ---- syntax/FB_Syntax_PropertiesFull.TcPOU
FUNCTION_BLOCK FB_Syntax_PropertiesFull
VAR
    _fPosition : LREAL;
    _bEnabled  : BOOL;
    _sDevName  : STRING(80);
END_VAR

PROPERTY Enabled : BOOL
GET
Enabled := _bEnabled;
END_GET
SET
_bEnabled := Enabled;
END_SET
END_PROPERTY

PROPERTY Position : LREAL
GET
Position := _fPosition;
END_GET
SET
IF Position >= 0.0 THEN
    _fPosition := Position;
END_IF
END_SET
END_PROPERTY

END_FUNCTION_BLOCK

// ---- syntax/FB_Syntax_PropertySet.TcPOU
FUNCTION_BLOCK FB_Syntax_PropertySet
VAR
    _nStored : INT;
END_VAR

_nStored := P_Value;

PROPERTY P_Value : INT
GET
P_Value := _nStored;
END_GET
SET
_nStored := P_Value;
END_SET
END_PROPERTY

END_FUNCTION_BLOCK

// ---- syntax/FB_Syntax_QueryInterface.TcPOU
FUNCTION_BLOCK FB_Syntax_QueryInterface
VAR
    ipWidget      : I_Syntax_Widget;
    ipExtended    : I_Syntax_Extended;
    fbDerived     : FB_Syntax_Derived;
    bHasExtended  : BOOL;
    bQuerySuccess : BOOL;
    hrResult      : hresult;
END_VAR

ipWidget := fbDerived;

IF ipWidget <> 0 THEN
    bQuerySuccess := __QUERYINTERFACE(ipWidget, ipExtended);

    IF bQuerySuccess AND (ipExtended <> 0) THEN
        bHasExtended := ipExtended.M_Execute(nCommand := 1);
    END_IF
END_IF

END_FUNCTION_BLOCK

// ---- syntax/FB_Syntax_StweepDisable.TcPOU
FUNCTION_BLOCK FB_Syntax_StweepDisable
VAR
    nA : INT;
    nB : INT;
END_VAR

nA := 1;

{stweep.disable}
nA := 99;
nB := 88;
{stweep.enable}
(* @stweep.disable *)
nA := 77;
(* @stweep.enable *)

nB := 2;

END_FUNCTION_BLOCK

// ---- syntax/FB_Syntax_SuperThis.TcPOU
FUNCTION_BLOCK FB_Syntax_SuperThis EXTENDS FB_Syntax_Derived
VAR
    _nLocal          : INT;
    _nExtendedStatus : INT;
END_VAR

SUPER^.M_Init();
_nLocal          := THIS^.M_GetValue();
_nExtendedStatus := THIS^.P_ExtendedStatus;

END_FUNCTION_BLOCK

// ---- syntax/FB_Syntax_VarInOut.TcPOU
FUNCTION_BLOCK FB_Syntax_VarInOut
VAR_INPUT
    nFactor : INT := 1;
END_VAR
VAR_IN_OUT
    nCounter : INT;
END_VAR
VAR
    _stLocal  : ST_Syntax_Mini;
    _nScratch : INT;
END_VAR

_nScratch      := nCounter * nFactor;
nCounter       := _nScratch;
_stLocal.nId   := nCounter;
_stLocal.sName := 'Updated';

METHOD M_Process : INT
VAR_INPUT
    nDelta : INT;
END_VAR
VAR_INST
    _nInstanceCounter : INT;
END_VAR
_nInstanceCounter := _nInstanceCounter + nDelta;
M_Process         := _nInstanceCounter;
END_METHOD

END_FUNCTION_BLOCK

// ---- syntax/FB_Syntax_WrapLongCall.TcPOU
FUNCTION_BLOCK FB_Syntax_WrapLongCall
VAR
    sA   : STRING(80);
    sB   : STRING(80);
    sC   : STRING(80);
    sD   : STRING(80);
    sE   : STRING(80);
    sOut : STRING(255);
    bOk  : BOOL;
END_VAR

bOk := FindAndReplace(
        pSrcString    := ADR(sA),
        pDeleteString := ADR(sB),
        pInsertString := ADR(sC),
        pDstString    := ADR(sD),
        nDstSize      := SIZEOF(sD));

IF bOk THEN
    sOut := CONCAT(CONCAT(CONCAT(sA, sB), sC), CONCAT(sD, sE));
END_IF

END_FUNCTION_BLOCK
